METHOD copyCmds : BOOL
VAR_IN_OUT 
	r_slaveArmCtrlCmd :ST_SlaveArmCtrlCmds;
END_VAR
r_slaveArmCtrlCmd.m_jntEnableFlag :=m_jntEnableFlag;
r_slaveArmCtrlCmd.m_cmdCartPose:=m_cmdCartPose;
r_slaveArmCtrlCmd.m_cmdCartTwist:=m_cmdCartTwist;
r_slaveArmCtrlCmd.m_simJntPos:=m_simJntPos;
r_slaveArmCtrlCmd.m_cmdJntPos:=m_cmdJntPos;
r_slaveArmCtrlCmd.m_cmdJntVel:=m_cmdJntVel;
r_slaveArmCtrlCmd.m_cmdJntAcc:=m_cmdJntAcc;
r_slaveArmCtrlCmd.m_cmdJntTrq:=m_cmdJntTrq;
r_slaveArmCtrlCmd.m_jntOPMode:=m_jntOPMode;
r_slaveArmCtrlCmd.m_FFJntTrq:=m_FFJntTrq;
END_METHOD

// call this function to add friction compensation to m_cmdJntTrq
METHOD enableFrictionCompensation : BOOL
VAR_IN_OUT CONSTANT
	i_slaveArm :FB_SlaveArm;
END_VAR

VAR
	i:INT;
	frictionScale :LREAL;
END_VAR
// add joint friction compensation
FOR i:=1 TO g_sJntNum DO
	frictionScale :=LIMIT(-1.0, i_slaveArm.curJntVel[i]/g_fullFrictionVel,1.0);
	m_cmdJntTrq[i]:=m_cmdJntTrq[i]+frictionScale * g_frictionCompScale * GVL_SlaveArmDynamics.g_slaveJntFriction[i_slaveArm.armIdx, i];
END_FOR
END_METHOD

// override this function in each exact controller
// NOTICE: set joint control mode here, and do some initialization if needed
METHOD PUBLIC init : BOOL
VAR_IN_OUT CONSTANT
	i_slaveArm	:FB_SlaveArm;
END_VAR
VAR_IN_OUT 
	r_slaveArmCtrlCmd :ST_SlaveArmCtrlCmds;
END_VAR
m_timePeriod:=0;
m_jntEnableFlag :=g_onesVec8i;
m_jntOPMode:=g_slaveAllPosMode;
m_cmdCartPose:=i_slaveArm.curCartPose;
m_cmdCartTwist:=g_zeroVec6d;
IF FALSE = m_holdLastCmds THEN
	m_cmdJntPos:=i_slaveArm.curJntPos;
ELSE
	m_cmdJntPos:=r_slaveArmCtrlCmd.m_cmdJntPos;
END_IF
m_simJntPos := m_cmdJntPos;
m_cmdJntVel:=g_zeroVec8d;
m_cmdJntAcc:=g_zeroVec8d;
m_cmdJntTrq:=g_zeroVec8d;
m_FFJntTrq :=g_zeroVec8d;

// update commands to arm
copyCmds(r_slaveArmCtrlCmd);
END_METHOD

PROPERTY isFinished : BOOL
GET
isFinished:=m_isFinished;
END_GET
END_PROPERTY

{warning '添加方法实现'}
METHOD reset : BOOL
m_isFinished:=FALSE;
m_timePeriod:=0;
END_METHOD

{warning '添加方法实现'}
METHOD run : BOOL
VAR_IN_OUT CONSTANT
	i_endoscopePose : ST_Frame;
	i_masterStatus :ST_MasterStatus;
	i_setupStatus: ST_SetupStatus;
	i_slaveArm :FB_SlaveArm;
END_VAR
VAR_IN_OUT
	r_slaveArmCtrlCmd :ST_SlaveArmCtrlCmds;
END_VAR
VAR
	i:INT;
END_VAR
IF m_isFinished THEN
	RETURN;
END_IF

// check if arm enabled
IF FALSE = i_slaveArm.isEnabled(m_jntEnableFlag) THEN
	RETURN;
END_IF

// calculate command joint position--Motion control
calcCmdJntPos(i_endoscopePose, i_masterStatus, i_setupStatus, i_slaveArm);

// calculate command joint torque -- Force control
calcCmdJntTrq(i_endoscopePose, i_masterStatus, i_setupStatus, i_slaveArm);

// update commands to arm
copyCmds(r_slaveArmCtrlCmd);

// update time period
m_timePeriod := m_timePeriod+g_slaveArmCtrlCycleTime;
END_METHOD

PROPERTY timePeriod : Lreal
GET
timePeriod := m_timePeriod;
END_GET
END_PROPERTY

END_FUNCTION_BLOCK

// ---- FBs_SlaveControllers/FB_SlaveCtrlInit.TcPOU
// Brief: Slave Arm Init
FUNCTION_BLOCK PUBLIC FB_SlaveCtrlInit EXTENDS FB_SlaveArmCtrlBase
VAR_INPUT
END_VAR
VAR_OUTPUT
END_VAR
VAR
	m_initState :INT :=0;
	
	// SDO writer
	m_MotorCurrentSDOWrite: ARRAY[1..5] OF FB_EcCoESdoWrite;
	// power box joint motor rated current
	m_wristJntRatedCurrent : DINT := 200;
END_VAR

// override this function in each exact controller
METHOD PROTECTED calcCmdJntPos : BOOL
VAR_IN_OUT CONSTANT
	i_endoscopePose : ST_Frame;
	i_masterStatus :ST_MasterStatus;
	i_setupStatus: ST_SetupStatus;
	i_slaveArm :FB_SlaveArm;
END_VAR

VAR 
	jntIdx:INT;
	SDOSubIndexCur :WORD;
	armIdx:INT;
END_VAR
IF m_timePeriod > 1.0 THEN
	m_isFinished := TRUE;
END_IF

// reset instrument control box motor current limit
armIdx :=i_slaveArm.armIdx;
FOR jntIdx :=4 TO 8 DO
	//动力盒移动关节和器械旋转关节，共享一个控制字，由SDO写入
	IF (jntIdx=8)  THEN
		SDOSubIndexCur:=16#6098;
	//动力盒3、5号电机为一个驱动器，共享一个控制字，由SDO写入
	ELSIF (jntIdx=4) OR (jntIdx=6)  THEN
		SDOSubIndexCur:=16#6099;
	//动力盒2、4号电机为一个驱动器，共享一个控制字，由SDO写入
	ELSIF (jntIdx=5) OR (jntIdx=7)  THEN
		SDOSubIndexCur:=16#609A;
	END_IF

	// write max motor current if it changes and works in position mode  GVL_SlaveMotorParameters.g_motorMaxCurrent[jntIdx]
	m_MotorCurrentSDOWrite[jntIdx-3](sNetID:= GVL_SlaveJointEncoderCaliData.g_slaveArmNetID[armIdx],
					nSlaveAddr := GVL_SlaveJointEncoderCaliData.g_slaveJointNetPort[armIdx,jntIdx],
					nSubIndex:=0,nIndex:=SDOSubIndexCur,pSrcBuf:=ADR(m_wristJntRatedCurrent),
					cbBufLen:=SIZEOF(m_wristJntRatedCurrent),bExecute:=TRUE);
	IF NOT m_MotorCurrentSDOWrite[jntIdx-3].bBusy THEN
		m_MotorCurrentSDOWrite[jntIdx-3](bExecute:=FALSE);
	END_IF
	
END_FOR
END_METHOD

METHOD PUBLIC init : BOOL
VAR_IN_OUT CONSTANT
	i_slaveArm	:FB_SlaveArm;
END_VAR
VAR_IN_OUT 
	r_slaveArmCtrlCmd :ST_SlaveArmCtrlCmds;
END_VAR

VAR
	i:INT;
END_VAR
SUPER^.Init(i_slaveArm,r_slaveArmCtrlCmd);
m_jntEnableFlag:=g_zeroVec8i;

// update commands to arm
copyCmds(r_slaveArmCtrlCmd);
END_METHOD

END_FUNCTION_BLOCK

// ---- FBs_SlaveControllers/FB_SlaveCtrlSelfCheck.TcPOU
// Brief: Slave Arm Run Self-check Trajectory
FUNCTION_BLOCK PUBLIC FB_SlaveCtrlSelfCheck EXTENDS FB_SlaveArmCtrlBase
VAR CONSTANT
	m_selfCheckMotionNum :INT :=1;
END_VAR
VAR
	// slave self-check motion parameters
	m_selfCheckPosture:ARRAY [1..m_selfCheckMotionNum, 1..g_sJntNum] OF LREAL:=[0.0, 	-PI/2, GVL_SlaveMotorParameters.g_maxDHJntPos[3], 	5(-g_2pi)];																			//PI/4, -PI/4, 0.3, pi, pi, pi, pi, pi];
	m_selfCheckMaxjntVel:Vec8d:=[0.2, 0.2, 0.1, 5(2.0)];
	m_selfCheckMaxjntAcc:Vec8d:=[1.0, 1.0, 0.5, 5(4.0)];
	m_selfCheckMaxjntJerk:Vec8d:=[2.0,2.0, 1.0, 5(8.0)];
	
	m_selfCheckTrajIdx: INT := 1;
	m_slefCheckPlanner: ARRAY[1..m_selfCheckMotionNum] OF FB_TrajMoveJ;
	
   // wait time for joint enable
   m_enableWaitTime :LREAL := 1.0;

   // time gap between enable and motion
   m_jntMotionTimeGap :LREAL := 0.5;

	
END_VAR

// override this function in each exact controller
METHOD PROTECTED calcCmdJntPos : BOOL
VAR_IN_OUT CONSTANT
	i_endoscopePose : ST_Frame;
	i_masterStatus :ST_MasterStatus;
	i_setupStatus: ST_SetupStatus;
	i_slaveArm :FB_SlaveArm;
END_VAR

VAR 
	i :INT;
	curJntVel :Vec8d;
END_VAR
// check if planner is ready
IF m_slefCheckPlanner[m_selfCheckTrajIdx].isGene = FALSE THEN
	calcCmdJntPos:=FALSE;
	RETURN;
END_IF

// arms enable successively
IF m_timePeriod > m_enableWaitTime THEN
       m_jntEnableFlag :=g_onesVec8i;
END_IF

IF m_timePeriod < m_enableWaitTime + m_jntMotionTimeGap THEN
	RETURN;
END_IF

// traj plan
calcCmdJntPos :=m_slefCheckPlanner[m_selfCheckTrajIdx].evaluate(m_timePeriod-m_enableWaitTime-m_jntMotionTimeGap, jntPos=> m_cmdJntPos, jntVel=>m_cmdJntVel, jntAcc=> m_cmdJntAcc);

// check if to transit to next segment
curJntVel :=i_slaveArm.curJntVel;
IF(m_timePeriod - m_enableWaitTime - m_jntMotionTimeGap > m_slefCheckPlanner[m_selfCheckTrajIdx].duration  AND norm(curJntVel)<7*GVL_SlaveControlParameters.g_jntStaticVelThres) THEN
	m_selfCheckTrajIdx:=m_selfCheckTrajIdx+1;
	m_timePeriod:=0;
END_IF

// check if to terminated
IF(m_selfCheckTrajIdx > m_selfCheckMotionNum) THEN
	m_isFinished:=TRUE;
END_IF
END_METHOD

METHOD PUBLIC init : BOOL
VAR_IN_OUT CONSTANT
	i_slaveArm	:FB_SlaveArm;
END_VAR
VAR_IN_OUT 
	r_slaveArmCtrlCmd :ST_SlaveArmCtrlCmds;
END_VAR

VAR
	i,j :INT;
	startJntPos,endJntPos :Vec8d;
	baseJntPos:Vec8d;
	cycleNum :LREAL;
END_VAR
SUPER^.Init(i_slaveArm,r_slaveArmCtrlCmd);
//m_jntEnableFlag :=g_zeroVec8i;

//set different wait time for each arm, so the arms would run self-check successively
m_enableWaitTime := i_slaveArm.armIdx-1;

// determine base joint position for instrument joint
baseJntPos :=g_zeroVec8d;
FOR i:=4 TO g_sJntNum DO
	cycleNum := FLOOR(i_slaveArm.curJntPos[i]/g_2pi);
	baseJntPos[i]:=cycleNum* g_2Pi;
END_FOR

// traj plan
// fisrt segment
// TODO: joint1/2 stay still in case arms collision
m_selfCheckTrajIdx :=1;
startJntPos:=i_slaveArm.curJntPos;
endJntPos:=startJntPos;
FOR j:=3 TO g_sJntNum DO 
	endJntPos[j]:=baseJntPos[j]+m_selfCheckPosture[1,j];
END_FOR
m_slefCheckPlanner[1].init(startJntPos,endJntPos,m_selfCheckMaxjntVel, m_selfCheckMaxjntAcc,m_selfCheckMaxjntJerk);

// other segments
IF m_selfCheckMotionNum>= 2 THEN
	FOR i:=2 TO m_selfCheckMotionNum DO 
		FOR j:=1 TO 7 DO 
			startJntPos[j]:=baseJntPos[j]+m_selfCheckPosture[i-1,j];
			endJntPos[j]:=baseJntPos[j]+m_selfCheckPosture[i,j];
		END_FOR
		m_slefCheckPlanner[i].init(startJntPos,endJntPos,m_selfCheckMaxjntVel, m_selfCheckMaxjntAcc,m_selfCheckMaxjntJerk);
	END_FOR
END_IF;

// update commands to arm
copyCmds(r_slaveArmCtrlCmd);
END_METHOD

END_FUNCTION_BLOCK

// ---- FBs_TrajectoryPlanning/FB_TrajMoveJ.TcPOU
FUNCTION_BLOCK FB_TrajMoveJ EXTENDS FB_TrajBase
VAR_OUTPUT
END_VAR
VAR
	// move vector in joint space
	m_startPos:Vec8d;
	m_targetPos:Vec8d;
	m_moveDir : Vec8d;
	m_moveDistance :LREAL;
	
	// doubleS planning for move distance
	m_doubleS :FB_BasicDoubleS;
END_VAR

METHOD evaluate : BOOL
VAR_INPUT
	t :LREAL;
END_VAR

VAR_OUTPUT
	jntPos,jntVel, jntAcc :vec8d;
END_VAR
VAR
	q,q_dot,q_ddot :LREAL;
	moveRange :Vec8d;
END_VAR
evaluate:=m_doubleS.evaluate(t,q=>q,q_dot=>q_dot, q_ddot=>q_dot);
IF evaluate =FALSE THEN
	RETURN;
END_IF

vecMultiNum(m_moveDir,q, moveRange);
vecAdd(moveRange, m_startPos,jntPos);
vecMultiNum(m_moveDir,q_dot, jntVel);
vecMultiNum( m_moveDir,q_ddot, jntAcc);
END_METHOD

METHOD init : BOOL
VAR_INPUT
	i_startJntPos :Vec8d;
	i_targetJntPos :Vec8d;
	i_maxJntVel : Vec8d;
	i_maxJntAcc : Vec8d;
	i_maxJntJerk :Vec8d;
END_VAR
VAR 
	i:INT;
	maxV, maxA, maxJ :LREAL;
	q:ARRAY[1..2] OF LREAL;
	v:ARRAY[1..2] OF LREAL;
END_VAR
m_startPos:=i_startJntPos;
m_targetPos:=i_targetJntPos;
vecSub(i_targetJntPos, i_startJntPos, m_moveDir);
m_moveDistance := norm(m_moveDir);

IF(m_moveDistance<g_smallNum) THEN
	vecMultiNum(g_onesVec7d,1/8, m_moveDir);;
ELSE
	vecMultiNum( m_moveDir,1/m_moveDistance, m_moveDir);
END_IF

// determian max vel/acc/jerk
maxV:=g_largeNum;
maxA:=g_largeNum;
maxJ:=g_largeNum;
FOR i :=1 TO 7 DO 
	IF ABS(m_moveDir[i])>g_smallNum THEN
		maxV := MIN (maxV, ABS(i_maxJntVel[i]/m_moveDir[i]));
		maxA := MIN (maxA, ABS(i_maxJntAcc[i]/m_moveDir[i]));
		maxJ := MIN (maxJ, ABS(i_maxJntJerk[i]/m_moveDir[i]));
	END_IF
END_FOR

// planning for moving distance
q[1]:=0;
q[2]:=m_moveDistance;
v[1]:=0;
v[2]:=0;
m_doubleS.init(q,v, maxV, maxA, maxJ);
m_duration:=m_doubleS.duration;
m_isGenerated:=m_doubleS.isGene;
END_METHOD

END_FUNCTION_BLOCK

// ---- FBs_SlaveControllers/FB_SlaveCtrlStandBy.TcPOU
// Brief: Slave Arm Standby
FUNCTION_BLOCK PUBLIC FB_SlaveCtrlStandBy EXTENDS FB_SlaveArmCtrlBase
VAR_INPUT
END_VAR
VAR_OUTPUT
END_VAR
VAR
END_VAR

METHOD PUBLIC init : BOOL
VAR_IN_OUT CONSTANT
	i_slaveArm	:FB_SlaveArm;
END_VAR
VAR_IN_OUT 
	r_slaveArmCtrlCmd :ST_SlaveArmCtrlCmds;
END_VAR
//init
SUPER^.Init(i_slaveArm,r_slaveArmCtrlCmd);
END_METHOD

END_FUNCTION_BLOCK

// ---- FBs_SlaveControllers/FB_SlaveCtrlMountPanel.TcPOU
// Brief: Mounting Panel
FUNCTION_BLOCK PUBLIC FB_SlaveCtrlMountPanel EXTENDS FB_SlaveArmCtrlBase
VAR_INPUT
END_VAR
VAR_OUTPUT
END_VAR
VAR
	// mount status
	m_mountStatus :INT := 0;
	
	// flag if joint is mounted
	m_jointMounted :ARRAY[1..5] OF BOOL := [5(FALSE)];
	
	// mount motion planning
	m_jntOTG :ARRAY[1..5] OF FB_secOrdTrajFilter;
	m_panelMountVel :LREAL := 2*pi;
	m_panelMountAcc :LREAL := 4*pi;
	
	// joint current threshold which indicate motor is buckled with panel
	m_maxJntCurrent :INT := 80;
	
	// command mount motion
	m_mountStepPos :LREAL := 45.0 * g_deg2Rad;
	m_targetMountPos :Vec5d;
	
	//panel clamp error Id
	m_panelClampErrId : UINT;
	m_panelClampTime : LREAL;
	m_noCurrentTime : LREAL :=10;
	m_notReturnToZero : LREAL :=15;
END_VAR

// override this function in each exact controller
METHOD PROTECTED calcCmdJntPos : BOOL
VAR_IN_OUT CONSTANT
	i_endoscopePose : ST_Frame;
	i_masterStatus :ST_MasterStatus;
	i_setupStatus: ST_SetupStatus;
	i_slaveArm :FB_SlaveArm;
END_VAR

VAR 
	i :INT;
	curJntPos :Vec8d;
	jntPosErr :Vec8d;
	cycleNum :LREAL;
END_VAR
IF m_panelClampErrId>0 THEN
	RETURN;
END_IF

curJntPos := i_slaveArm.curJntPos;

CASE m_mountStatus OF
	// To lock joint with panel
	0:
		FOR i:=1 TO 5 DO
			// check joint buckled with panel
			IF ABS(i_slaveArm.filtJntCurrent[i+3])> m_maxJntCurrent THEN 
				m_jointMounted[i]:=TRUE;
				m_targetMountPos[i]:=curJntPos[i+3];
				m_jntOTG[i].init(m_targetMountPos[i], 0,m_panelMountVel, m_panelMountAcc, g_slaveArmCtrlCycleTime);
			END_IF
			
			// set command joint position step
			IF FALSE = m_jointMounted[i] THEN
				m_targetMountPos[i]:=curJntPos[i+3]+m_mountStepPos;
			END_IF
		END_FOR
		
		IF (m_jointMounted[1] AND m_jointMounted[2] AND m_jointMounted[3] AND m_jointMounted[4] AND m_jointMounted[5]) or m_timePeriod > 5.0 THEN
			m_mountStatus:=1;
		END_IF
	
	// determine zero position
	1:
		FOR i:=1 TO 5 DO
			cycleNum := FLOOR(curJntPos[i+3]/g_2pi);
			m_targetMountPos[i]:=cycleNum* g_2Pi;
		END_FOR
		m_mountStatus :=2;
	
	// move back to zero position
	2:
		m_isFinished:=TRUE;
		FOR i:=1 TO 5 DO
			IF ABS(m_targetMountPos[i]-curJntPos[i+3])>GVL_SlaveControlParameters.g_jntCtrlAngTolHigh THEN
				m_isFinished:=FALSE;
				EXIT;
			END_IF
		END_FOR
END_CASE

//panel clamp status check
m_panelClampErrId := panelClampStatus();

// traj plan
FOR i:=1 TO 5 DO
	m_jntOTG[i].run(m_targetMountPos[i],0.0, o_cmdAcc=>m_cmdJntAcc[3+i],o_cmdVel=>m_cmdJntVel[3+i],o_cmdPos=>m_cmdJntPos[i+3]);
END_FOR
END_METHOD

METHOD PUBLIC init : BOOL
VAR_IN_OUT CONSTANT
	i_slaveArm	:FB_SlaveArm;
END_VAR
VAR_IN_OUT 
	r_slaveArmCtrlCmd :ST_SlaveArmCtrlCmds;
END_VAR
VAR
	i : INT;
END_VAR
SUPER^.Init(i_slaveArm,r_slaveArmCtrlCmd);
m_jntOPMode[4] := DriverOPMode_PosTrq;
m_jntOPMode[5] := DriverOPMode_PosTrq;
m_jntOPMode[6] := DriverOPMode_PosTrq;
m_jntOPMode[7] := DriverOPMode_PosTrq;
m_jntOPMode[8] := DriverOPMode_PosTrq;

m_mountStatus:=0;
FOR i:=1 TO 5 DO
	m_targetMountPos[i]:=m_cmdJntPos[i+3];
	m_jntOTG[i].init(m_targetMountPos[i], 0,m_panelMountVel, m_panelMountAcc, g_slaveArmCtrlCycleTime);
	m_jointMounted[i]:=FALSE;
END_FOR
m_panelClampTime :=0;
m_panelClampErrId := 0;
// update commands to arm
copyCmds(r_slaveArmCtrlCmd);
END_METHOD

PROPERTY panelClampErrId : UINT
GET
panelClampErrId := m_panelClampErrId;
END_GET
END_PROPERTY

METHOD panelClampStatus : UINT
VAR_IN_OUT CONSTANT
END_VAR
//m_panelClampErrId=1 panel clamp the current does not reach the set value
//m_panelClampErrId=2 panel clamp position does not return to zero
m_panelClampTime := LIMIT(0,m_panelClampTime + g_slaveArmCtrlCycleTime,10);

IF m_mountStatus=0  AND m_panelClampTime>=m_noCurrentTime  THEN
	panelClampStatus := 1;
ELSIF m_mountStatus=2 AND m_panelClampTime>=m_notReturnToZero  THEN
	panelClampStatus := 2;
END_IF
END_METHOD

END_FUNCTION_BLOCK

// ---- FBs_SlaveControllers/FB_SlaveCtrlPanelReady.TcPOU
// Brief: Panel Ready
FUNCTION_BLOCK PUBLIC FB_SlaveCtrlPanelReady EXTENDS FB_SlaveArmCtrlBase
VAR_INPUT
END_VAR
VAR_OUTPUT
END_VAR
VAR
END_VAR

// override this function in each exact controller
// NOTICE: set joint control mode here, and do some initialization if needed
METHOD PUBLIC init : BOOL
VAR_IN_OUT CONSTANT
	i_slaveArm	:FB_SlaveArm;
END_VAR
VAR_IN_OUT 
	r_slaveArmCtrlCmd :ST_SlaveArmCtrlCmds;
END_VAR
//init
SUPER^.Init(i_slaveArm,r_slaveArmCtrlCmd);

//update the control mode ---1028
m_jntOPMode := g_slaveAllPosMode;
m_jntOPMode[1]:=DriverOPMode_PosTrq;
m_jntOPMode[2]:=DriverOPMode_PosTrq;

copyCmds(r_slaveArmCtrlCmd);
END_METHOD

END_FUNCTION_BLOCK

// ---- FBs_SlaveControllers/FB_SlaveCtrlMountInstru.TcPOU
// Brief: Mounting Instrument
FUNCTION_BLOCK PUBLIC FB_SlaveCtrlMountInstru EXTENDS FB_SlaveArmCtrlBase
VAR
	// mount status
	m_instruMountStatus :INT := 0;
	m_scopeMountStatus :INT := 0;
	m_ultrasoundMountStatus :INT :=0 ;
	
	// flag if joint is mounted
	m_jointMounted :ARRAY[1..5] OF BOOL := [5(FALSE)];
	
	// instrument mount motion range
	m_mountMotionAng :Vec5d :=[5(pi)];
	
	// instrument mount direction
	m_mountDir :Vec5i :=[1, 1, 1, 1, 1];
	
	// mount motion planning
	m_jntOTG :ARRAY[1..5] OF FB_secOrdTrajFilter;
	m_instruMountVel :LREAL := 4*PI;
	m_instruMountAcc :LREAL := 8*PI;
	
	//Joint 4 half-range angle of instrument
	m_instruJnt4HalfRangeAng :LREAL := 323*g_deg2Rad;
	
	// joint current threshold which indicate panel is buckled with instrument
	m_maxJntCurrent :Vec5d := [150, 150, 150, 180, 180];
	
	// command mount motion
	m_targetMountPos :Vec8d;
	
	// instrument zero position
	m_instruZeroDeviation :Vec5d;
	
	//ultrasound knife Reduce the current rotation Angle  J3
	m_ultraKnifeRotaAngleJ3 :LREAL := 30*g_deg2Rad;
	
	// ultrasound knife rotate angle zero position
	m_ultraKnifeRotAngZeroPos :LREAL := 4.50567;
	
	// joint position error
	m_jntPosErr :Vec5d;
	
	// endoscope motion angle to original position
	m_scopeJnt4CenterMotionAng :LREAL :=175*g_deg2Rad;
	m_scopeJnt5CenterMotionAng :LREAL :=150*g_deg2Rad;
	
	//instrument clamp error Id
	m_instruClampErrId : UINT;
	m_instruClampTime : LREAL;
	m_noCurrentTime : LREAL :=3;
	m_notReturnToZero : LREAL :=5;
END_VAR

// override this function in each exact controller
METHOD PROTECTED calcCmdJntPos : BOOL
VAR_IN_OUT CONSTANT
	i_endoscopePose : ST_Frame;
	i_masterStatus :ST_MasterStatus;
	i_setupStatus: ST_SetupStatus;
	i_slaveArm :FB_SlaveArm;
END_VAR

VAR 
END_VAR
// mount error detect;
m_instruClampErrId := instruClampStatus(i_slaveArm);

// return directly if instrument/endoscope is not readed
IF NOT(i_slaveArm.instrument.onChipData.m_InstruReadSucceed) THEN
	return;
END_IF

IF i_slaveArm.instrument.onChipData.m_InstruReadSucceed AND InstruType_endoscope = i_slaveArm.instrument.onChipData.m_InstruID THEN
	mountEndoscope(i_slaveArm);
ELSIF i_slaveArm.instrument.onChipData.m_InstruReadSucceed AND InstruType_NewEndoscope = i_slaveArm.instrument.onChipData.m_InstruID THEN
	mountNewEndoscope(i_slaveArm);
ELSIF i_slaveArm.instrument.onChipData.m_InstruReadSucceed AND (InstruType_UltrasoundKnifeS = i_slaveArm.instrument.m_instruType OR InstruType_UltrasoundKnifeU = i_slaveArm.instrument.m_instruType) THEN
	mountUltraKnife(i_slaveArm);
ELSE
	mountInstrument(i_slaveArm);
END_IF
END_METHOD

METHOD PUBLIC init : BOOL
VAR_IN_OUT CONSTANT
	i_slaveArm	:FB_SlaveArm;
END_VAR
VAR_IN_OUT 
	r_slaveArmCtrlCmd :ST_SlaveArmCtrlCmds;
END_VAR

VAR
	i : INT;
END_VAR
// check if to hold the command joint position unchanged
m_holdLastCmds := checkToHoldLastCmds(i_slaveArm);

SUPER^.Init(i_slaveArm,r_slaveArmCtrlCmd);
m_jntOPMode[4] := DriverOPMode_PosTrq;
m_jntOPMode[5] := DriverOPMode_PosTrq;
m_jntOPMode[6] := DriverOPMode_PosTrq;
m_jntOPMode[7] := DriverOPMode_PosTrq;
m_jntOPMode[8] := DriverOPMode_PosTrq;

FOR i:=1 TO 5 DO
	m_targetMountPos[i+3]:=m_cmdJntPos[i+3];
	m_jntOTG[i].init(m_targetMountPos[i+3], 0,m_instruMountVel, m_instruMountAcc, g_slaveArmCtrlCycleTime);
	m_jointMounted[i]:=FALSE;
END_FOR

m_instruMountStatus:=0;
m_scopeMountStatus:=0;
m_ultrasoundMountStatus:=0;
m_instruClampErrId := 0;
m_instruClampTime := 0;
// update commands to arm
copyCmds(r_slaveArmCtrlCmd);
END_METHOD

PROPERTY instruClampErrId :  UINT
GET
instruClampErrId := m_instruClampErrId;
END_GET
END_PROPERTY

METHOD instruClampStatus : UINT
VAR_IN_OUT CONSTANT
	i_slaveArm :FB_SlaveArm;
END_VAR
//m_instruClampErrId=1 instrumen clamp the current does not reach the set value
//m_instruClampErrId=2 instrumen clamp position does not return to zero
m_instruClampTime := LIMIT(0,m_instruClampTime + g_slaveArmCtrlCycleTime,10);
IF i_slaveArm.instrument.onChipData.m_InstruReadSucceed THEN
	IF InstruType_endoscope = i_slaveArm.instrument.m_instruType THEN
		IF (m_scopeMountStatus=0 OR m_scopeMountStatus=1) AND m_instruClampTime>=m_noCurrentTime  THEN
			instruClampStatus := 1;
		ELSIF m_scopeMountStatus=3 AND m_instruClampTime>=m_notReturnToZero  THEN
			instruClampStatus := 2;
		END_IF
		
	ELSIF (InstruType_UltrasoundKnifeS = i_slaveArm.instrument.m_instruType OR InstruType_UltrasoundKnifeU = i_slaveArm.instrument.m_instruType) THEN
		IF (m_ultrasoundMountStatus=0) AND m_instruClampTime>=m_noCurrentTime  THEN
			instruClampStatus := 1;
		ELSIF (m_scopeMountStatus=3) AND m_instruClampTime>=m_notReturnToZero  THEN
			instruClampStatus := 2;
		END_IF
			
	ELSE
		IF (m_instruMountStatus=0) AND m_instruClampTime>=m_noCurrentTime  THEN
			instruClampStatus := 1;
		ELSIF (m_instruMountStatus=3) AND m_instruClampTime>=m_notReturnToZero  THEN
			instruClampStatus := 2;
		END_IF
	END_IF
END_IF
END_METHOD

METHOD mountEndoscope : BOOL
VAR_IN_OUT CONSTANT
	i_slaveArm :FB_SlaveArm;
END_VAR

VAR 
	i :INT;
	curJntPos :Vec8d;
END_VAR
curJntPos := i_slaveArm.curJntPos;

CASE m_scopeMountStatus OF
	//fix scope lock joint(joint 7)
	0:
		// other joints stay still
		FOR i:=1 TO 3 DO
			m_jointMounted[i] := TRUE;
			m_targetMountPos[i+3]:=curJntPos[i+3];
			m_jntOTG[i].init(m_targetMountPos[i+3], 0,m_instruMountVel, m_instruMountAcc, g_slaveArmCtrlCycleTime);
		END_FOR
	
		// check if buckled
		m_jointMounted[4]:=FALSE; 
		m_jointMounted[5]:=FALSE; 
		IF ABS(i_slaveArm.filtJntCurrent[7])> m_maxJntCurrent[4] THEN 
			m_jointMounted[4]:=TRUE;
			m_targetMountPos[7]:=curJntPos[7];
			m_jntOTG[4].init(m_targetMountPos[7], 0,m_instruMountVel, m_instruMountAcc, g_slaveArmCtrlCycleTime);
			m_scopeMountStatus:=1;
		ELSE
			m_targetMountPos[7]:=curJntPos[7]+m_mountMotionAng[4];
		END_IF

	1: // buckle scope rotate joint (joint 8)
		m_jointMounted[5]:=FALSE; 
		IF ABS(i_slaveArm.filtJntCurrent[8])> m_maxJntCurrent[5] THEN 
			m_jointMounted[5]:=TRUE;
			m_targetMountPos[8]:=curJntPos[8];
			m_jntOTG[5].init(m_targetMountPos[8], 0,m_instruMountVel, m_instruMountAcc, g_slaveArmCtrlCycleTime);
			m_scopeMountStatus:=2;
		ELSE
			m_targetMountPos[8]:=curJntPos[8]+m_mountMotionAng[5];
		END_IF
	

	2:// move back to zero position
		m_targetMountPos[7]:= curJntPos[7]-m_scopeJnt4CenterMotionAng;
		m_targetMountPos[8]:= curJntPos[8]-m_scopeJnt5CenterMotionAng;
		m_scopeMountStatus :=3;
		
		
	3:
		IF ABS(m_targetMountPos[7]-curJntPos[7]) <GVL_SlaveControlParameters.g_jntCtrlAngTolHigh AND 
				ABS(m_targetMountPos[8]-curJntPos[8]) <GVL_SlaveControlParameters.g_jntCtrlAngTolHigh THEN
			// record current joint position as offset for instrument
			i_slaveArm.instrument.initInstruJntPos(i_slaveArm.curJntPos);
			m_isFinished := TRUE;
		END_IF
		
END_CASE

// traj plan
FOR i:=1 TO 5 DO
	m_jntOTG[i].run(m_targetMountPos[i+3],0.0, o_cmdAcc=>m_cmdJntAcc[3+i],o_cmdVel=>m_cmdJntVel[3+i],o_cmdPos=>m_cmdJntPos[i+3]);
END_FOR
END_METHOD

METHOD mountInstrument : BOOL
VAR_IN_OUT CONSTANT
	i_slaveArm :FB_SlaveArm;
END_VAR

VAR 
	i :INT;
	curJntPos :Vec8d;
END_VAR
curJntPos := i_slaveArm.curJntPos;

// joint4 stay still if instrument has only on finger
IF i_slaveArm.instrument.instruTypeInfo.m_isSingleFinger THEN
	m_jointMounted[1]:=TRUE;
END_IF

CASE m_instruMountStatus OF
	// To lock panel with instrument
	0:
		//buckle panel with instrument
		FOR i:=1 TO 4 DO
			// check if buckled 
			IF ABS(i_slaveArm.filtJntCurrent[i+3])> m_maxJntCurrent[i] AND ABS(i_slaveArm.curJntVel[i+3])<1.0*g_deg2Rad THEN 
				m_jointMounted[i]:=TRUE;
				m_targetMountPos[i+3]:=curJntPos[i+3];
				m_jntOTG[i].init(m_targetMountPos[i+3], 0,m_instruMountVel, m_instruMountAcc, g_slaveArmCtrlCycleTime);
			END_IF
			
			// set target joint position
			IF FALSE = m_jointMounted[i] THEN
				IF i = 4 THEN
					m_targetMountPos[i+3]:=curJntPos[i+3]+m_mountMotionAng[i];
				ELSE
					m_targetMountPos[i+3]:=curJntPos[i+3]-m_mountMotionAng[i];
				END_IF
				
			END_IF
		END_FOR
		
		
		// check transition condition
		IF (m_jointMounted[1] AND m_jointMounted[2] AND m_jointMounted[3] AND m_jointMounted[4])  THEN
			IF i_slaveArm.instrument.onChipData.m_InstruReadSucceed THEN//Check whether the data is read successfully
				m_instruMountStatus:=1;
			END_IF
		END_IF
	
	1:// calculation deviates from the instrument zero position
		FOR i:=1 TO 4 DO
			m_instruZeroDeviation[i] :=  i_slaveArm.linkSingle[i+3] - i_slaveArm.instrument.onChipData.m_InstruPos[i];
		END_FOR
		m_instruMountStatus :=2;
	
	
	2:// move back to zero position
		FOR i:=1 TO 3 DO//J1-3
			IF m_instruZeroDeviation[i]>pi THEN
				m_instruZeroDeviation[i] := m_instruZeroDeviation[i] - 2*PI;
			ELSIF m_instruZeroDeviation[i]<-pi THEN
				m_instruZeroDeviation[i] := m_instruZeroDeviation[i] + 2*PI;
			END_IF
		END_FOR
		
		//joint4
		IF m_instruZeroDeviation[4]>0 AND m_instruZeroDeviation[4] < pi THEN
			m_instruZeroDeviation[4] := m_instruZeroDeviation[4] - 2*pi;
		ELSIF m_instruZeroDeviation[4]<0 AND m_instruZeroDeviation[4] > -pi THEN
			m_instruZeroDeviation[4] := m_instruZeroDeviation[4] + 2*pi;
		END_IF
		
		// set target joint position
		FOR i:=1 TO 4 DO
			m_targetMountPos[i+3]:=curJntPos[i+3] - m_instruZeroDeviation[i];
		END_FOR
		m_instruMountStatus :=3;
	
	3: // move to zero position
		m_instruMountStatus :=4;
		FOR i:=1 TO 4 DO 
			m_jntPosErr[i]:=m_targetMountPos[i+3]-curJntPos[i+3];
			IF ABS(m_jntPosErr[i]) >GVL_SlaveControlParameters.g_jntCtrlAngTolLow OR 
					ABS( i_slaveArm.linkSingle[i+3] - i_slaveArm.instrument.onChipData.m_InstruPos[i]) >5*g_deg2rad THEN
				m_instruMountStatus :=3;
				EXIT;
			END_IF
		END_FOR
	
	4:
		// record current joint position as offset for instrument
		i_slaveArm.instrument.initInstruJntPos(i_slaveArm.curJntPos);
		
		m_isFinished :=  TRUE;

END_CASE

// traj plan
FOR i:=1 TO 4 DO
	m_jntOTG[i].run(m_targetMountPos[i+3],0.0, o_cmdAcc=>m_cmdJntAcc[3+i],o_cmdVel=>m_cmdJntVel[3+i],o_cmdPos=>m_cmdJntPos[i+3]);
END_FOR
END_METHOD

METHOD mountNewEndoscope : BOOL
VAR_IN_OUT CONSTANT
	i_slaveArm :FB_SlaveArm;
END_VAR

VAR 
	i :INT;
	curJntPos :Vec8d;
END_VAR
curJntPos := i_slaveArm.curJntPos;

CASE m_scopeMountStatus OF
	//fix scope lock joint(joint 7)
	0:
		// other joints stay still
		FOR i:=1 TO 5 DO
			IF i = 1 OR i =2 OR i =5 THEN
				m_jointMounted[i] := TRUE;
				m_targetMountPos[i+3]:=curJntPos[i+3];
				m_jntOTG[i].init(m_targetMountPos[i+3], 0,m_instruMountVel, m_instruMountAcc, g_slaveArmCtrlCycleTime);
			END_IF
		END_FOR
	
		// check if buckled
		m_jointMounted[3]:=FALSE; 
		m_jointMounted[4]:=FALSE; 
		FOR i:=3 TO 4 DO
			IF ABS(i_slaveArm.filtJntCurrent[i+3])> m_maxJntCurrent[i] THEN 
				m_jointMounted[i]:=TRUE;
				m_targetMountPos[i+3]:=curJntPos[i+3];
				m_jntOTG[i].init(m_targetMountPos[i+3], 0,m_instruMountVel, m_instruMountAcc, g_slaveArmCtrlCycleTime);
				
			ELSE
				m_targetMountPos[i+3]:=curJntPos[i+3]+m_mountMotionAng[i];
			END_IF
		END_FOR
		
		IF m_jointMounted[3] AND m_jointMounted[4] THEN
			m_scopeMountStatus:=1;
		END_IF
		

	1: // buckle scope rotate joint (joint 8)
		m_jntOPMode[6] := DriverOPMode_Trq;
		m_instruZeroDeviation[4] :=  i_slaveArm.linkSingle[7] - i_slaveArm.instrument.onChipData.m_InstruPos[4];
		m_scopeMountStatus :=2;

	2:// move back to zero position
		
		//joint4
		IF m_instruZeroDeviation[4]>0 AND m_instruZeroDeviation[4] > pi THEN
			m_instruZeroDeviation[4] := m_instruZeroDeviation[4] - 2*pi;
		ELSIF m_instruZeroDeviation[4]<0 AND m_instruZeroDeviation[4] < -pi THEN
			m_instruZeroDeviation[4] := m_instruZeroDeviation[4] + 2*pi;
		END_IF
		
		m_targetMountPos[7]:=curJntPos[7] - m_instruZeroDeviation[4];
		m_scopeMountStatus :=3;
		
		
	3:
		m_isFinished := FALSE;
		IF ABS(m_targetMountPos[7]-curJntPos[7]) <GVL_SlaveControlParameters.g_jntCtrlAngTolHigh THEN
			// record current joint position as offset for instrument
			i_slaveArm.instrument.initInstruJntPos(i_slaveArm.curJntPos);
			m_isFinished := TRUE;
		END_IF
		
END_CASE

// traj plan
FOR i:=1 TO 5 DO
	m_jntOTG[i].run(m_targetMountPos[i+3],0.0, o_cmdAcc=>m_cmdJntAcc[3+i],o_cmdVel=>m_cmdJntVel[3+i],o_cmdPos=>m_cmdJntPos[i+3]);
END_FOR

// joint6 output torque to help rotation motion
IF m_jntOPMode[6] = DriverOPMode_Trq THEN
	m_cmdJntTrq[6] := -0.5*i_slaveArm.cmdJntTrq[7];
END_IF
END_METHOD

METHOD mountUltraKnife : BOOL
VAR_IN_OUT CONSTANT
	i_slaveArm :FB_SlaveArm;
END_VAR

VAR 
	i :INT;
	curJntPos :Vec8d;
END_VAR
curJntPos := i_slaveArm.curJntPos;

m_jointMounted[1]:=TRUE;
m_jointMounted[2]:=TRUE;


CASE m_ultrasoundMountStatus OF 
	// To lock panel with instrument
	0:
		//buckle panel with instrument
		FOR i:=3 TO 5 DO
			// check if buckled 
			IF ABS(i_slaveArm.filtJntCurrent[i+3])> m_maxJntCurrent[i] THEN 
				m_jointMounted[i]:=TRUE;
				m_targetMountPos[i+3]:=curJntPos[i+3];
				m_jntOTG[i].init(m_targetMountPos[i+3], 0,m_instruMountVel, m_instruMountAcc, g_slaveArmCtrlCycleTime);
			END_IF
			
			// set target joint position
			IF FALSE = m_jointMounted[i] THEN
				IF i = 5 THEN
					m_targetMountPos[i+3]:=curJntPos[i+3]+m_mountMotionAng[i];
				ELSE
					m_targetMountPos[i+3]:=curJntPos[i+3]-m_mountMotionAng[i];
				END_IF
				
			END_IF
		END_FOR

		// check transition condition
		IF ( m_jointMounted[3] AND m_jointMounted[4] AND m_jointMounted[5] )  THEN
			IF i_slaveArm.instrument.onChipData.m_InstruReadSucceed THEN//Check whether the data is read successfully
				m_ultrasoundMountStatus:=1;
			END_IF
		END_IF

	1:
		//m_jntOPMode[8] := DriverOPMode_Trq;
		// calculation deviates from the instrument zero position
		m_instruZeroDeviation[3] :=   i_slaveArm.linkSingle[6] - i_slaveArm.instrument.onChipData.m_InstruPos[3]; //m_ultraKnifeRotaAngleJ3;
		m_instruZeroDeviation[4] :=  i_slaveArm.linkSingle[7] - m_ultraKnifeRotAngZeroPos;
		m_ultrasoundMountStatus :=2;
		
	2:// move back to zero position
		//joint3
		IF m_instruZeroDeviation[3] > 2*pi THEN
			m_instruZeroDeviation[3] := m_instruZeroDeviation[3] - 2*pi  ;
		ELSIF  m_instruZeroDeviation[3] < -pi THEN
			m_instruZeroDeviation[3] := 2*pi + m_instruZeroDeviation[3] ;
		END_IF
		//joint4
		IF m_instruZeroDeviation[4]>0 AND m_instruZeroDeviation[4] < pi THEN
			m_instruZeroDeviation[4] := m_instruZeroDeviation[4] - 2*pi;
		ELSIF m_instruZeroDeviation[4]<0 AND m_instruZeroDeviation[4] > -pi THEN
			m_instruZeroDeviation[4] := m_instruZeroDeviation[4] + 2*pi;
		END_IF
	
		// set target joint position
		m_targetMountPos[6]:=curJntPos[6] - m_instruZeroDeviation[3];
		m_targetMountPos[7]:=curJntPos[7] - m_instruZeroDeviation[4];
		m_targetMountPos[8]:=curJntPos[8] - m_instruZeroDeviation[4];

		m_ultrasoundMountStatus :=3;

	3:
		// joint8 in passive mode
		m_jntOPMode[8] := DriverOPMode_Trq;
		
		m_isFinished:=TRUE;
		FOR i:=3 TO 4 DO 
			m_jntPosErr[i]:=m_targetMountPos[i+3]-curJntPos[i+3];
			IF ABS(m_jntPosErr[i]) >GVL_SlaveControlParameters.g_jntCtrlAngTolLow  THEN
				m_isFinished := FALSE;
				EXIT;
			END_IF
		END_FOR	
		
		// record current joint position as offset for instrument
		i_slaveArm.instrument.initInstruJntPos(i_slaveArm.curJntPos);

END_CASE


// traj plan
FOR i:=1 TO 5 DO
	m_jntOTG[i].run(m_targetMountPos[i+3],0.0, o_cmdAcc=>m_cmdJntAcc[3+i],o_cmdVel=>m_cmdJntVel[3+i],o_cmdPos=>m_cmdJntPos[i+3]);
END_FOR
END_METHOD

END_FUNCTION_BLOCK

// ---- FBs_SlaveControllers/FB_SlaveCtrlInstruReady.TcPOU
// Brief: Instrument Ready
FUNCTION_BLOCK PUBLIC FB_SlaveCtrlInstruReady EXTENDS FB_SlaveArmCtrlBase
VAR_INPUT
END_VAR
VAR_OUTPUT
END_VAR
VAR
END_VAR

METHOD PUBLIC init : BOOL
VAR_IN_OUT CONSTANT
	i_slaveArm	:FB_SlaveArm;
END_VAR
VAR_IN_OUT 
	r_slaveArmCtrlCmd :ST_SlaveArmCtrlCmds;
END_VAR


VAR
	j:INT;
	maxJntErr:LREAL;
	jntCtrlErr:Vec7d;
END_VAR
//NOTE:DO NOT hold last command

//init
SUPER^.Init(i_slaveArm,r_slaveArmCtrlCmd);
END_METHOD

END_FUNCTION_BLOCK

// ---- FBs_SlaveControllers/FB_SlaveCtrlMasterSlave.TcPOU
// Brief: Slave Arm MasterSlave controller
FUNCTION_BLOCK PUBLIC FB_SlaveCtrlMasterSlave EXTENDS FB_SlaveArmCtrlBase
VAR
	// pose track control kp
	m_posTrackKp :REAL := 0;
	m_oriTrackKp :REAL := 100;
	
	// minimum distance between instrument tip and remote center
	m_minInstruRCDis:LREAL := 0.05;
	
	// master-slave motion scale
	m_MSMotionScale :LREAL;
		
	// gripper match angle threshold
	m_gripperMatchAngThres :LREAL := 2*g_deg2Rad;
	
	// control error thershold from joint limit back to free space
	m_jntLimitOriErr :LREAL :=g_deg2Rad * 5;
	
	// master-slave error thershold to halt control 
	m_safetyOriErr :LREAL :=g_deg2Rad * 150;
	
	// filter cut-off frequency for master-slave control
	m_macroCmdJntPosLpfCutoffFreq : LREAL :=5;
	m_microCmdJntPosLpfCutoffFreq : LREAL :=15;
	
	// last command joint position
	m_lastCmdJntPos :Vec8d;
	
	// simulated DH joint position
	m_simDHJntPos : Vec6d;
	
	// simulated slave twist of DH joint
	m_simDHJointVel :Vec6d;
		
	// enter master-slave control for the first time
	m_firstIn :BOOL := TRUE;
	
	// flag if reach joint limit
	m_reachMacroJntLimit :BOOL;
	m_reachWristJntLimit :BOOL;
	m_jntLimitFlag :Vec6b;
	
	// master/slave origin pose when first enter master-slave control
	m_masterOriginPose : ST_Frame;
	m_slaveOriginPose : ST_Frame;
	
	// orientation deviation(in master coordinate) between master and slave when first enter control
	m_MSOriDeviation : Mat3d;
	
	// command joint position filter
	m_cmdJntPosLpf:ARRAY[1..8] OF FB_LowPassFilter;
	
	// commmand yaw angle and velocity
	m_cmdYawAngle :LREAL;
	m_cmdYawVel :LREAL;
	
	// comand yaw angle and velocity filter
	m_cmdYawAngLpf : FB_LowPassFilter;
	m_cmdYawVelLpf : FB_LowPassFilter;
	
	// master pose/velocity in monitor coordinate
	m_masterPose :ST_Frame;
	m_masterTwist : Vec6d;
	
	// master grip angle
	m_masterGripAngle : LREAL;
	
	// slave command/current pose in endoscope coordinate
	m_slaveCmdPoseInScope :ST_Frame;
	m_slavePoseInScope : ST_Frame;
	
	// slave command/current pose in cart
	m_slaveCmdPoseInCart :ST_Frame;
	m_slavePoseInCart : ST_Frame;
	
	// instrument controller
	m_basicInstruController : FB_BasicInstruControl;
	m_usKnifeController : FB_UltrosonicKnifeControl;
	
	// slave command grip angle and grip force level
	m_slaveCmdGripAngle :LREAL;
	m_slaveCmdGripForceLevel:LREAL;
	
	// slave pose error
	m_slavePosErr :Vec3d;
	m_slaveRotErr :Mat3d;
	m_errAngle : LREAL;
	m_errAxisLocal, m_errAxis :Vec3d;
	m_masterSlavePoseError :Vec6d;
	
	// master velocity in slave coordinate
	m_masterFFVel, m_masterFFWVel :Vec3d;
	
	// velocity for slave to track master motion
	m_slaveCmdVel, m_slaveCmdWVel : Vec3d;
	
	// flag to start gripper control
	m_gripperCtrlFlag :BOOL;
	
	// instrument tyep
	m_instruType : E_InstrumentType;
	
	//################# variable to interpolate master pose ##############
	m_firstInterpolate :BOOL :=TRUE;
	m_lastMasterPose : ST_Frame;
	m_lastMasterGripAngle :LREAL;
	m_masterInterpolateCycle :INT := 4;
	m_curInterpolateCylce :INT := 1;
	m_masterPosInterStep :Vec3d;
	m_masterOriInterStep :Mat3d;
	m_masterGripAngleInterStep :LREAL;
	m_interplotedMasterPose :ST_Frame;
	m_interplotedMasterGripAngle :LREAL;
	
	// code execute time measure
	m_codeTime : Profiler;
	
	
END_VAR

METHOD PROTECTED calcCmdJntPos : BOOL
VAR_IN_OUT CONSTANT
	i_endoscopePose : ST_Frame;
	i_masterStatus :ST_MasterStatus;
	i_setupStatus: ST_SetupStatus;
	i_slaveArm :FB_SlaveArm;
END_VAR

VAR 
	i,j : INT;
	tmpMat3d : Mat3d;
	masterMotionRange : Vec3d;
	
	masterVelInScope, masterWVelInScope :Vec3d;
	masterVelInCart, masterWVelInCart :Vec3d;

	cmdVelScale :LREAL;
	invJaco :Mat6d;
	armJntJaco,armJntJacoInv, wristJntJaco :Mat3d;
	velByWristJnt,velByArmJnt : Vec3d;
	armDHJntVel, wristDHJntVel :Vec3d;
	tmpFrame : ST_Frame;
	jnt3Limit :LREAL;
	jntDynaUB, jntDynaLB :LREAL;
END_VAR
m_codeTime(START:=TRUE, RESET:=TRUE);

IF isFinished THEN
	RETURN;
END_IF

// decide matched master arm index
FOR i:=1 TO g_mArmNum DO 
	IF i_masterStatus.m_teleSlaveArmIdx[i] = i_slaveArm.armIdx THEN
		masterPoseInterploate(i_masterStatus.m_curArmPose[i],i_masterStatus.m_gripAngle[i], i_slaveArm);
		m_masterPose := m_interplotedMasterPose;
		m_masterGripAngle := m_interplotedMasterGripAngle;
		m_masterTwist := i_masterStatus.m_curArmTwist[i];
	END_IF
END_FOR

// compute slave pose in endoscope coordinate
m_slavePoseInCart := transform(i_setupStatus.m_curEndPose[i_slaveArm.armIdx], i_slaveArm.simCartPose);
tmpFrame :=invFrame(i_endoscopePose);
m_slavePoseInScope := transform(tmpFrame, m_slavePoseInCart);

// handle for the first time in
IF TRUE = m_firstIn THEN
	m_firstIn := FALSE;
	m_masterOriginPose :=m_masterPose;
	m_slaveOriginPose := m_slavePoseInScope;
	matTranspose(m_masterOriginPose.m_rot, tmpMat3d);
	matMultiply(tmpMat3d, m_slavePoseInScope.m_rot,m_MSOriDeviation);
	m_lastMasterGripAngle := m_masterGripAngle;
	
	// only update motion scale while entering teleControl 
	m_MSMotionScale := 1.0/ MAX(1,  i_masterStatus.m_motionScale);
END_IF

// compute master twist in slave arm coordinate
FOR i:=1 TO 3 DO
	masterVelInScope[i] := m_masterTwist[i]*m_MSMotionScale;
	masterWVelInScope[i] := m_masterTwist[i+3];
END_FOR
matMultiVec(i_endoScopePose.m_rot, masterVelInScope, masterVelInCart);
matMultiVec(i_endoScopePose.m_rot, masterWVelInScope, masterWVelInCart);
matTranspose(i_setupStatus.m_curEndPose[i_slaveArm.armIdx].m_rot, tmpMat3d);
matMultiVec(tmpMat3d,masterVelInCart, m_masterFFVel);
matMultiVec(tmpMat3d,masterWVelInCart, m_masterFFWVel);

// compute slave command pose in scope
vecSub(m_masterPose.m_pos, m_masterOriginPose.m_pos, masterMotionRange);
vecSelfMultiNum(masterMotionRange, m_MSMotionScale);
vecAdd(m_slaveOriginPose.m_pos, masterMotionRange, m_slaveCmdPoseInScope.m_pos);
matMultiply(m_masterPose.m_rot, m_MSOriDeviation, m_slaveCmdPoseInScope.m_rot);

// compute slave command pose in slave arm coordinate
m_slaveCmdPoseInCart := transform(i_endoScopePose, m_slaveCmdPoseInScope);
tmpFrame := invFrame(i_setupStatus.m_curEndPose[i_slaveArm.armIdx]);
m_cmdCartPose := transform(tmpFrame, m_slaveCmdPoseInCart);

// compute pose error
vecSub(m_cmdCartPose.m_pos, i_slaveArm.simCartPose.m_pos, m_slavePosErr);
matTranspose(i_slaveArm.simCartPose.m_rot, tmpMat3d);
matMultiply(tmpMat3d, m_cmdCartPose.m_rot, m_slaveRotErr);
rot2AngAxis(m_slaveRotErr, angle=>m_errAngle, axis=>m_errAxisLocal);
matMultiVec(i_slaveArm.simCartPose.m_rot, m_errAxisLocal, m_errAxis);

// calculate pose error in endoscope
calcMSErrInScope(i_endoscopePose, i_setupStatus.m_curEndPose[i_slaveArm.armIdx], i_slaveArm);

//safety check
IF ABS(m_errAngle)>m_safetyOriErr THEN
	m_isFinished := TRUE;
	RETURN;
END_IF

// pose track control
vecMultiNum(m_slavePosErr, m_posTrackKp, m_slaveCmdVel);
vecMultiNum(m_errAxis, m_errAngle*m_oriTrackKp, m_slaveCmdWVel);
// final command twist
FOR i:=1 TO 3 DO 
	m_cmdCartTwist[i] := m_slaveCmdVel[i] + m_masterFFVel[i];
	m_cmdCartTwist[i+3] := m_slaveCmdWVel[i] + m_masterFFWVel[i];
END_FOR

// compute command velocity for DH joints
invJaco := i_slaveArm.simJacoInv;
matMultiVec(invJaco, m_cmdCartTwist, m_simDHJointVel);

// limit instrument wrist dofs
limitInstruDofs(i_slaveArm, m_simDHJointVel);

// limit instrument wrist joint velocity
wristLimitSolve(i_slaveArm);

// limit DH joints velocity 
FOR i:=4 TO 6 DO 
	m_simDHJointVel[i] := LIMIT(-GVL_SlaveMotorParameters.g_maxJntVel[i], m_simDHJointVel[i], GVL_SlaveMotorParameters.g_maxJntVel[i]);
END_FOR

// modify arm joints velocity to compensate wrist joint motion
FOR i:=1 TO 3 DO
	FOR j:=1 TO 3 DO
		armJntJaco[i,j]:=i_slaveArm.simJaco[i,j];
		wristJntJaco[i,j]:=i_slaveArm.simJaco[i,j+3];
	END_FOR
	armDHJntVel[i]:=m_simDHJointVel[i];
	wristDHJntVel[i]:=m_simDHJointVel[i+3];
	m_slaveCmdVel[i] := m_cmdCartTwist[i];
END_FOR
invMat3(armJntJaco, armJntJacoInv);
matMultiVec(wristJntJaco, wristDHJntVel, velByWristJnt);
vecSub(m_slaveCmdVel, velByWristJnt, velByArmJnt);
matMultiVec(armJntJacoInv, velByArmJnt, armDHJntVel);

// limit arm joint position
m_reachMacroJntLimit:=false;
FOR i:=1 TO 3 DO
	IF i=3 THEN
		jnt3Limit := i_slaveArm.instrument.instruTypeInfo.m_rodLength+i_slaveArm.instrument.instruTypeInfo.m_headLength - GVL_SlaveArmKinematic.g_minInstruRCDis;
		jntDynaUB := MAX( 0, (jnt3Limit - i_slaveArm.simDHJntPos[i])/g_slaveArmCtrlCycleTime);
	ELSE
		jntDynaUB := MAX( 0, (GVL_SlaveMotorParameters.g_maxDHJntPos[i] - i_slaveArm.simDHJntPos[i])/g_slaveArmCtrlCycleTime);
	END_IF
	jntDynaLB := MIN( 0, (GVL_SlaveMotorParameters.g_minDHJntPos[i] - i_slaveArm.simDHJntPos[i])/g_slaveArmCtrlCycleTime);
	
	IF m_simDHJointVel[i] >= jntDynaUB OR m_simDHJointVel[i]<= jntDynaLB THEN
		armDHJntVel[i]:=LIMIT(jntDynaLB, m_simDHJointVel[i], jntDynaUB);
		m_reachMacroJntLimit:=TRUE;
	END_IF
END_FOR

// limit DH joints velocity 
FOR i:=1 TO 3 DO
	m_simDHJointVel[i]:=armDHJntVel[i];
	m_simDHJointVel[i+3]:=wristDHJntVel[i];
END_FOR
cmdVelScale := 1;
FOR i:=1 TO g_cartDofs DO 
	cmdVelScale:=MAX(cmdVelScale, ABS(m_simDHJointVel[i]/GVL_SlaveMotorParameters.g_maxJntVel[i]));
END_FOR
vecSelfMultiNum(m_simDHJointVel, 1.0/cmdVelScale);

// integrate command DH joint position
FOR i:=1 TO 6 DO
	m_simDHJntPos[i] := i_slaveArm.simDHJntPos[i] + m_simDHJointVel[i]*g_slaveArmCtrlCycleTime;
END_FOR

// gripper angle/force control
gripperControl(i_slaveArm);

// calculate target motor joint position/velocity from DH joint position
i_slaveArm.instrument.instruIK(m_simDHJntPos,m_slaveCmdGripAngle, o_jntPos=>m_simJntPos);

// filt command joint position
FOR i:=1 TO g_sJntNum DO 
	m_cmdJntPos[i] := m_cmdJntPosLpf[i].run(m_simJntPos[i]);
END_FOR

// compute command joint velocity
vecSub(m_cmdJntPos, m_lastCmdJntPos, m_cmdJntVel);
vecSelfMultiNum(m_cmdJntVel, g_slaveArmCtrlFreq);
m_lastCmdJntPos:=m_cmdJntPos;

m_codeTime(START:=FALSE);
END_METHOD

// override this function in each exact controller
METHOD PROTECTED calcCmdJntTrq : BOOL
VAR_IN_OUT CONSTANT
	i_endoscopePose : ST_Frame;
	i_masterStatus :ST_MasterStatus;
	i_setupStatus: ST_SetupStatus;
	i_slaveArm :FB_SlaveArm;
END_VAR
VAR
	i :INT ;
	instruCmdGripAngle, instruCmdGripForceLevel :LREAL;
	instruCmdJntPos, instruCmdJntVel : Vec5d;	
	instruJntCtrlTrq :Vec5d;
END_VAR
IF isFinished THEN
	RETURN;
END_IF

// set joint torque to zero in default
m_cmdJntTrq := g_zeroVec8d;

// instrument joint control
FOR i:=1 TO 5 DO 
	instruCmdJntPos[i]:=m_cmdJntPos[i+3];
	instruCmdJntVel[i]:=m_cmdJntVel[i+3];
END_FOR
m_cmdYawAngle := m_cmdYawAngLpf.run(m_simDHJntPos[6]);
m_cmdYawVel := m_cmdYawVelLpf.run(m_simDHJointVel[6]);

// check if to exert larger grip force
setMaxGripTrq(i_masterStatus, i_slaveArm);


IF i_slaveArm.instrument.instruType = InstruType_UltrasoundKnifeS OR i_slaveArm.instrument.instruType = InstruType_UltrasoundKnifeU THEN
	m_usKnifeController.run(instruCmdJntPos,instruCmdJntVel, m_slaveCmdGripForceLevel, i_slaveArm, o_cmdJntTrq=>instruJntCtrlTrq);
ELSE
	m_basicInstruController.run(instruCmdJntPos,instruCmdJntVel, m_cmdYawAngle, m_cmdYawVel, m_slaveCmdGripForceLevel, i_slaveArm, o_cmdJntTrq=>instruJntCtrlTrq);
END_IF

FOR i:=1 TO 5 DO
	m_cmdJntTrq[i+3]:=instruJntCtrlTrq[i];
END_FOR
END_METHOD

METHOD calcMSErrInScope : BOOL
VAR_IN_OUT CONSTANT
	i_endoscopePose : ST_Frame;
	i_setupPose :ST_Frame;
	i_slaveArm :FB_SlaveArm;
END_VAR
VAR
	posErrInCart,oriErrInCart :Vec3d;
	invRot :Mat3d;
	posErrInScope,oriErrInScope :Vec3d;
	i:INT;
END_VAR
m_masterSlavePoseError := g_zeroVec6d;

// pose error caused by joints limits
IF m_reachMacroJntLimit THEN
	// pose error in cart coordinate
	matMultiVec(i_setupPose.m_rot, m_slavePosErr, posErrInCart);
	
	// pose err in endoscope coordinate
	matTranspose(i_endoscopePose.m_rot, invRot);
	matMultiVec(invRot, posErrInCart, posErrInScope);
	
	FOR i:=1 TO 3 DO 
		m_masterSlavePoseError[i]:=posErrInScope[i];
	END_FOR
END_IF

// pose error caused by joints limits
IF  m_reachWristJntLimit THEN
	// pose error in cart coordinate
	matMultiVec(i_setupPose.m_rot, m_errAxis, oriErrInCart);
	vecSelfMultiNum(oriErrInCart, m_errAngle);
	
	// pose err in endoscope coordinate
	matTranspose(i_endoscopePose.m_rot, invRot);
	matMultiVec(invRot, oriErrInCart, oriErrInScope);
	
	FOR i:=1 TO 3 DO 
		m_masterSlavePoseError[i+3]:=oriErrInScope[i];
	END_FOR
END_IF
END_METHOD

METHOD PUBLIC clearBacklash : BOOL
VAR_INPUT
END_VAR
m_basicInstruController.clearBacklash();
m_usKnifeController.clearBacklash();
END_METHOD

METHOD gripperControl : BOOL
VAR_IN_OUT CONSTANT
	i_slaveArm :FB_SlaveArm;
END_VAR

VAR
	matchedSlaveGripAngle:LREAL;
	matchedSlaveGripForce:LREAL;
	masterGripVelThres :LREAL := 5.0 *g_deg2Rad;
END_VAR
// compute matched slave grip angle and force
i_slaveArm.instrument.gripAngleMap(m_masterGripAngle,o_instruGripAngle=>matchedSlaveGripAngle, o_instruGripForceLevel=>matchedSlaveGripForce);

IF m_gripperCtrlFlag THEN
	m_slaveCmdGripAngle := matchedSlaveGripAngle;
	m_slaveCmdGripForceLevel := matchedSlaveGripForce;
	RETURN;
ELSE
	//m_gripperCtrlFlag := (ABS(m_masterGripAngleVel) >masterGripVelThres) AND  (m_masterGripAngleVel * (matchedSlaveGripAngle-i_slaveArm.curGripAngle)>0);
	m_gripperCtrlFlag := ABS(matchedSlaveGripAngle-i_slaveArm.curGripAngle)<m_gripperMatchAngThres OR 
	     (matchedSlaveGripAngle>=i_SlaveArm.instrument.instruTypeInfo.m_maxGripAngle - m_gripperMatchAngThres AND i_slaveArm.curGripAngle>=matchedSlaveGripAngle) OR 
		(matchedSlaveGripAngle<=g_minSlaveGripAngle + m_gripperMatchAngThres AND i_slaveArm.curGripAngle<=matchedSlaveGripAngle);
END_IF
END_METHOD

METHOD PUBLIC init : BOOL
VAR_IN_OUT CONSTANT
	i_slaveArm	:FB_SlaveArm;
END_VAR
VAR_IN_OUT 
	r_slaveArmCtrlCmd :ST_SlaveArmCtrlCmds;
END_VAR
VAR 
	i :INT ;
END_VAR
SUPER^.Init(i_slaveArm,r_slaveArmCtrlCmd);
m_simJntPos :=m_cmdJntPos;
m_lastCmdJntPos :=m_cmdJntPos;
m_jntOPMode[1] := DriverOPMode_PosTrq;
m_jntOPMode[2] := DriverOPMode_PosTrq;
m_jntOPMode[3] := DriverOPMode_PosTrq;
m_jntOPMode[4] := DriverOPMode_Trq;
m_jntOPMode[5] := DriverOPMode_Trq;
m_jntOPMode[6] := DriverOPMode_Trq;
m_jntOPMode[7] := DriverOPMode_Trq;
m_jntOPMode[8] := DriverOPMode_Trq;
m_firstIn :=TRUE;
m_gripperCtrlFlag :=FALSE;

// init gripper angle
m_slaveCmdGripAngle := i_slaveArm.curGripAngle;
m_slaveCmdGripForceLevel:=0;

// init filter
FOR i:=1 TO 3 DO
	m_cmdJntPosLpf[i].init(1, m_macroCmdJntPosLpfCutoffFreq, g_slaveArmCtrlFreq);
END_FOR
FOR i:=4 TO g_sJntNum DO
	m_cmdJntPosLpf[i].init(1, m_microCmdJntPosLpfCutoffFreq, g_slaveArmCtrlFreq);
END_FOR
m_cmdYawAngLpf.init(1, m_microCmdJntPosLpfCutoffFreq, g_slaveArmCtrlFreq);
m_cmdYawVelLpf.init(1, m_microCmdJntPosLpfCutoffFreq, g_slaveArmCtrlFreq);

// init controller
m_basicInstruController.init(i_slaveArm);
m_usKnifeController.init(i_slaveArm);
m_instruType := i_slaveArm.instrument.instruType;

// init interpolation data
m_firstInterpolate :=TRUE;
m_curInterpolateCylce := 1;

// update commands to arm
copyCmds(r_slaveArmCtrlCmd);
END_METHOD

PROPERTY InstruBacklash : Vec5d
GET
IF m_instruType = InstruType_UltrasoundKnifeS OR m_instruType = InstruType_UltrasoundKnifeU THEN
	instruBacklash := m_usKnifeController.m_jntBacklash;
ELSE
	instruBacklash := m_basicInstruController.m_jntBacklash;
END_IF
END_GET
END_PROPERTY

// limit specific joint dofs based on instrument types
METHOD PRIVATE limitInstruDofs : BOOL
VAR_IN_OUT CONSTANT
	i_slaveArm :FB_SlaveArm;
END_VAR

VAR_IN_OUT
	r_simDHJointVel :Vec6d;
END_VAR
IF i_slaveArm.instrument.instruType = InstruType_UltrasoundKnifeS OR i_slaveArm.instrument.instruType = InstruType_UltrasoundKnifeU THEN
	r_simDHJointVel[5] :=0;
	r_simDHJointVel[6] :=0;
END_IF
END_METHOD

// every some cycles the data from master robots would be miss, so add this interpolation
METHOD masterPoseInterploate : BOOL
VAR_IN_OUT CONSTANT
	i_masterPose :ST_FRAME;
	i_masterGripAngle :LREAL;
	i_slaveArm :FB_SlaveArm;
END_VAR

VAR
	rotT :Mat3d;
	rotErr:Mat3d;
	errAngle:LREAL;
	errAxisLocal :Vec3d;
	tmpMat :Mat3d;
	cartVel, DHJntVel :Vec6d;
	wVelWrd:Vec3d;
	i :INT;
	invJaco :Mat6d;
	cmdVelScale :LREAL;
END_VAR
IF m_firstInterpolate THEN
	m_firstInterpolate :=FALSE;
	m_lastMasterGripAngle :=i_masterGripAngle;
	m_lastMasterPose := i_masterPose;
	m_masterPosInterStep :=g_zeroVec3d;
	m_masterOriInterStep :=g_eye3d;
	m_masterGripAngleInterStep :=0.0;
	m_interplotedMasterPose := i_masterPose;
	m_interplotedMasterGripAngle := i_masterGripAngle;
END_IF


// update next interpolation
IF m_curInterpolateCylce > m_masterInterpolateCycle THEN
	vecSub(i_masterPose.m_pos, m_lastMasterPose.m_pos, m_masterPosInterStep);
	vecSelfMultiNum( m_masterPosInterStep, 1.0/INT_TO_LREAL(m_masterInterpolateCycle));
	
	matTranspose(m_lastMasterPose.m_rot, rotT);
	matMultiply(rotT, i_masterPose.m_rot, rotErr);
	rot2AngAxis(rotErr, angle=>errAngle, axis=>errAxisLocal);
	m_masterOriInterStep := angAxis2Rot(errAngle/INT_TO_LREAL(m_masterInterpolateCycle), errAxisLocal);
	
	// cap linear step based on macro joint velocity limit
	matMultiVec(i_slaveArm.simCartPose.m_rot, errAxisLocal, wVelWrd);
	vecSelfMultiNum(wVelWrd, errAngle*g_slaveArmCtrlFreq/INT_TO_LREAL(m_masterInterpolateCycle));
	FOR i:=1 TO 3 DO
		cartVel[i] := m_masterPosInterStep[i]*m_MSMotionScale*g_slaveArmCtrlFreq;
		cartVel[i+3] := wVelWrd[i];
	END_FOR
	invJaco := i_slaveArm.simJacoInv;
	matMultiVec(invJaco, cartVel, DHJntVel);
	cmdVelScale := 1;
	FOR i:=1 TO 3 DO 
		cmdVelScale:=MAX(cmdVelScale, ABS(DHJntVel[i]/GVL_SlaveMotorParameters.g_maxJntVel[i]));
	END_FOR
	vecSelfMultiNum(m_masterPosInterStep, 1.0/cmdVelScale);
	
	m_masterGripAngleInterStep := (i_masterGripAngle- m_lastMasterGripAngle)/INT_TO_LREAL(m_masterInterpolateCycle);
	
	m_curInterpolateCylce :=1;
	m_lastMasterPose:= i_masterPose;
	m_lastMasterGripAngle := i_masterGripAngle;
END_IF

// control points
IF m_curInterpolateCylce = m_masterInterpolateCycle THEN
	m_interplotedMasterGripAngle := m_lastMasterGripAngle;
	m_interplotedMasterPose.m_rot := m_lastMasterPose.m_rot;
ELSE
	m_interplotedMasterGripAngle := m_interplotedMasterGripAngle + m_masterGripAngleInterStep;
	vecSelfAdd(m_interplotedMasterPose.m_pos, m_masterPosInterStep);
	tmpMat := m_interplotedMasterPose.m_rot;
	matMultiply(tmpMat, m_masterOriInterStep, m_interplotedMasterPose.m_rot);
END_IF

m_curInterpolateCylce:= m_curInterpolateCylce+1;
END_METHOD

PROPERTY masterSlavePoseErr : REFERENCE to Vec6d
GET
masterSlavePoseErr REF= m_masterSlavePoseError;
END_GET
END_PROPERTY

METHOD setMaxGripTrq : BOOL
VAR_IN_OUT CONSTANT
	i_masterStatus :ST_MasterStatus;
	i_slaveArm :FB_SlaveArm;
END_VAR
VAR
	i:INT;
	 peakGripTrqScale :LREAL := 2;
END_VAR
// only valid for ForceBipolar
IF i_slaveArm.instrument.instruType <> InstruType_ForceBipolar THEN
	RETURN;
END_IF

// only trigger grip force switch when no grip force exerted currently
IF m_slaveCmdGripForceLevel > g_smallNum  THEN
	RETURN;
END_IF; 

// decide matched master arm index
FOR i:=1 TO g_mArmNum DO 
	IF i_masterStatus.m_teleSlaveArmIdx[i] = i_slaveArm.armIdx THEN
		IF i_masterStatus.m_pedalHover[i] AND i_masterStatus.m_electricKnifePedalTrigger[i] =1 THEN
		   m_basicInstruController.setMaxGripTrq(i_slaveArm.instrument.instruTypeInfo.m_normGripTrq * peakGripTrqScale);
		ELSE
		   m_basicInstruController.setMaxGripTrq(i_slaveArm.instrument.instruTypeInfo.m_normGripTrq);
		END_IF
	END_IF
END_FOR
END_METHOD

// calculate optimized wrist joint velocity when joint limit is violated
METHOD wristLimitSolve : BOOL
VAR_IN_OUT CONSTANT
	i_slaveArm :FB_SlaveArm;
END_VAR

VAR
	i,j:INT;
	jntDynaUB, jntDynaLB :LREAL;
	
	dsrWVel:Vec3d;
	wristJntVel :Vec3d;
	wristJaco:Mat3d;
	
	optJntVel:Vec2d;
	partJaco :Mat32;
	partJacoT :Mat23;
	JtJ,JtJInv :Mat2d;
	partJacoPInv:Mat23;
	
	partJacoPinv2 :Vec3d;
	jacoNorm :LREAL;
	
	wVelLocal,wVelWrd:Vec3d;
	matT:Mat3d;
END_VAR
m_reachWristJntLimit := FALSE;

// desire angular velocity from wrist joint
FOR i:=1 TO 3 DO
	wristJntVel[i] := m_simDHJointVel[i+3];
	FOR j:=1 TO 3 DO
		wristJaco[i,j]:= i_slaveArm.simJaco[i+3, j+3];
	END_FOR 
END_FOR
matMultiVec(wristJaco, wristJntVel, dsrWVel);

// check which joint reaches limit
FOR i:=4 TO 6 DO
	m_jntLimitFlag[i] := FALSE;
	jntDynaUB := MAX( 0, (i_slaveArm.instrument.m_wristMaxDHJntPos[i-3] - i_slaveArm.simDHJntPos[i])/g_slaveArmCtrlCycleTime);
	jntDynaLB := MIN( 0, (i_slaveArm.instrument.m_wristMinDHJntPos[i-3] - i_slaveArm.simDHJntPos[i])/g_slaveArmCtrlCycleTime);
	IF m_simDHJointVel[i] >= jntDynaUB OR m_simDHJointVel[i]<=jntDynaLB THEN
		m_simDHJointVel[i]:=LIMIT(jntDynaLB, m_simDHJointVel[i], jntDynaUB);
		m_jntLimitFlag[i]:=TRUE;
		m_reachWristJntLimit := TRUE;
	END_IF
END_FOR

// no limit violated
IF NOT( m_jntLimitFlag[4]) AND NOT(m_jntLimitFlag[5]) AND NOT(m_jntLimitFlag[6]) THEN
	RETURN;
END_IF; 

// all joint reach limit
IF m_jntLimitFlag[4] AND m_jntLimitFlag[5] AND m_jntLimitFlag[6] THEN
	RETURN;
END_IF;

// joint 4 reach limit
IF m_jntLimitFlag[4] AND NOT(m_jntLimitFlag[5]) AND NOT(m_jntLimitFlag[6]) THEN
	// colume 2/3
	partJaco[1,1]:= wristJaco[1,2];
	partJaco[2,1]:= wristJaco[2,2];
	partJaco[3,1]:= wristJaco[3,2];
	
	partJaco[1,2]:= wristJaco[1,3];
	partJaco[2,2]:= wristJaco[2,3];
	partJaco[3,2]:= wristJaco[3,3];
	
	// pinv partJaco
	matTranspose(partJaco, partJacoT);
	matMultiply(partJacoT, partJaco, JtJ);
	IF NOT(invMat2(JtJ, JtJInv)) THEN
		m_simDHJointVel[5] :=0;
		m_simDHJointVel[6] := 0;
		RETURN;
	END_IF
	matMultiply(JtJInv, partJacoT, partJacoPinv);
	
	// desire angular velocity exclusive limited joint motion
	dsrWVel[1] := dsrWVel[1] - wristJaco[1,1] * m_simDHJointVel[4];
	dsrWVel[2] := dsrWVel[2] - wristJaco[2,1] * m_simDHJointVel[4];
	dsrWVel[3] := dsrWVel[3] - wristJaco[3,1] * m_simDHJointVel[4];
	
	//NOTE: special handle for roll limit. avoiding joint5/6 motion caused by roll limit
	matTranspose(i_slaveArm.simCartPose.m_rot, matT);
	matMultiVec(matT, dsrWVel, wVelLocal);
	wVelLocal[3]:=0;
	matMultiVec(i_slaveArm.simCartPose.m_rot, wVelLocal, dsrWVel);
	
	// solve
	matMultiVec(partJacoPinv, dsrWVel, optJntVel);
	m_simDHJointVel[5] :=optJntVel[1];
	m_simDHJointVel[6] := optJntVel[2];
END_IF

// joint 5 reach limit
IF m_jntLimitFlag[5] AND NOT(m_jntLimitFlag[4]) AND NOT(m_jntLimitFlag[6]) THEN
	// colume 1/3
	partJaco[1,1]:= wristJaco[1,1];
	partJaco[2,1]:= wristJaco[2,1];
	partJaco[3,1]:= wristJaco[3,1];
	
	partJaco[1,2]:= wristJaco[1,3];
	partJaco[2,2]:= wristJaco[2,3];
	partJaco[3,2]:= wristJaco[3,3];
	
	// pinv partJaco
	matTranspose(partJaco, partJacoT);
	matMultiply(partJacoT, partJaco, JtJ);
	IF NOT(invMat2(JtJ, JtJInv)) THEN
		m_simDHJointVel[4] :=0;
		m_simDHJointVel[6] := 0;
		RETURN;
	END_IF
	matMultiply(JtJInv, partJacoT, partJacoPinv);
		
	// desire angular velocity exclusive limited joint motion
	dsrWVel[1] := dsrWVel[1] - wristJaco[1,2] * m_simDHJointVel[5];
	dsrWVel[2] := dsrWVel[2] - wristJaco[2,2] * m_simDHJointVel[5];
	dsrWVel[3] := dsrWVel[3] - wristJaco[3,2] * m_simDHJointVel[5];
	
	//NOTE: special handle for pitch limit. avoiding joint4/6 motion caused by pitch limit
	matTranspose(i_slaveArm.simCartPose.m_rot, matT);
	matMultiVec(matT, dsrWVel, wVelLocal);
	wVelLocal[1]:=0;
	matMultiVec(i_slaveArm.simCartPose.m_rot, wVelLocal, dsrWVel);
	
	// solve
	matMultiVec(partJacoPinv, dsrWVel, optJntVel);
	m_simDHJointVel[4] :=optJntVel[1];
	m_simDHJointVel[6] := optJntVel[2];
END_IF

// joint 6 reach limit
IF m_jntLimitFlag[6] AND NOT(m_jntLimitFlag[4]) AND NOT(m_jntLimitFlag[5]) THEN
	// colume 1/2
	partJaco[1,1]:= wristJaco[1,1];
	partJaco[2,1]:= wristJaco[2,1];
	partJaco[3,1]:= wristJaco[3,1];
	
	partJaco[1,2]:= wristJaco[1,2];
	partJaco[2,2]:= wristJaco[2,2];
	partJaco[3,2]:= wristJaco[3,2];
	
	// pinv partJaco
	matTranspose(partJaco, partJacoT);
	matMultiply(partJacoT, partJaco, JtJ);
	IF NOT(invMat2(JtJ, JtJInv)) THEN
		m_simDHJointVel[4] :=0;
		m_simDHJointVel[5] := 0;
		RETURN;
	END_IF
	matMultiply(JtJInv, partJacoT, partJacoPinv);
		
	// desire angular velocity exclusive limited joint motion
	dsrWVel[1] := dsrWVel[1] - wristJaco[1,3] * m_simDHJointVel[6];
	dsrWVel[2] := dsrWVel[2] - wristJaco[2,3] * m_simDHJointVel[6];
	dsrWVel[3] := dsrWVel[3] - wristJaco[3,3] * m_simDHJointVel[6];
	
	// solve
	matMultiVec(partJacoPinv, dsrWVel, optJntVel);
	m_simDHJointVel[4] :=optJntVel[1];
	m_simDHJointVel[5] := optJntVel[2];
END_IF

// joint 4/5 reach limit
IF m_jntLimitFlag[4] AND m_jntLimitFlag[5] AND NOT(m_jntLimitFlag[6]) THEN
	// pinv partJaco of column 3
	partJacoPinv2[1] := wristJaco[1, 3];
	partJacoPinv2[2] := wristJaco[2, 3];
	partJacoPinv2[3] := wristJaco[3, 3];
	jacoNorm := norm(partJacoPinv2);
	vecSelfMultiNum(partJacoPinv2, 1.0/(jacoNorm*jacoNorm));
		
	// desire angular velocity exclusive limited joint motion
	dsrWVel[1] := dsrWVel[1] - wristJaco[1,1] * m_simDHJointVel[4] - wristJaco[1,2] * m_simDHJointVel[5];
	dsrWVel[2] := dsrWVel[2] - wristJaco[2,1] * m_simDHJointVel[4] - wristJaco[2,2] * m_simDHJointVel[5];
	dsrWVel[3] := dsrWVel[3] - wristJaco[3,1] * m_simDHJointVel[4] - wristJaco[3,2] * m_simDHJointVel[5];
	
	// solve
	m_simDHJointVel[6] := vecDot(partJacoPinv2, dsrWVel);
END_IF

// joint 4/6 reach limit
IF m_jntLimitFlag[4] AND m_jntLimitFlag[6] AND NOT(m_jntLimitFlag[5]) THEN
	// pinv partJaco of column 2
	partJacoPinv2[1] := wristJaco[1, 2];
	partJacoPinv2[2] := wristJaco[2, 2];
	partJacoPinv2[3] := wristJaco[3, 2];
	jacoNorm := norm(partJacoPinv2);
	vecSelfMultiNum(partJacoPinv2, 1.0/(jacoNorm*jacoNorm));
		
	// desire angular velocity exclusive limited joint motion
	dsrWVel[1] := dsrWVel[1] - wristJaco[1,1] * m_simDHJointVel[4] - wristJaco[1,3] * m_simDHJointVel[6];
	dsrWVel[2] := dsrWVel[2] - wristJaco[2,1] * m_simDHJointVel[4] - wristJaco[2,3] * m_simDHJointVel[6];
	dsrWVel[3] := dsrWVel[3] - wristJaco[3,1] * m_simDHJointVel[4] - wristJaco[3,3] * m_simDHJointVel[6];
	
	// solve
	m_simDHJointVel[5] := vecDot(partJacoPinv2, dsrWVel);
END_IF

// joint 5/6 reach limit
IF m_jntLimitFlag[5] AND m_jntLimitFlag[6] AND NOT(m_jntLimitFlag[4]) THEN
	// pinv partJaco of column 4
	partJacoPinv2[1] := wristJaco[1, 1];
	partJacoPinv2[2] := wristJaco[2, 1];
	partJacoPinv2[3] := wristJaco[3, 1];
	jacoNorm := norm(partJacoPinv2);
	vecSelfMultiNum(partJacoPinv2, 1.0/(jacoNorm*jacoNorm));
		
	// desire angular velocity exclusive limited joint motion
	dsrWVel[1] := dsrWVel[1] - wristJaco[1,2] * m_simDHJointVel[5] - wristJaco[1,3] * m_simDHJointVel[6];
	dsrWVel[2] := dsrWVel[2] - wristJaco[2,2] * m_simDHJointVel[5] - wristJaco[2,3] * m_simDHJointVel[6];
	dsrWVel[3] := dsrWVel[3] - wristJaco[3,2] * m_simDHJointVel[5] - wristJaco[3,3] * m_simDHJointVel[6];
	
	// solve
	m_simDHJointVel[4] := vecDot(partJacoPinv2, dsrWVel);
END_IF


// check which joint reaches limit
FOR i:=4 TO 6 DO
	jntDynaUB := MAX( 0, (i_slaveArm.instrument.m_wristMaxDHJntPos[i-3] - i_slaveArm.simDHJntPos[i])/g_slaveArmCtrlCycleTime);
	jntDynaLB := MIN( 0, (i_slaveArm.instrument.m_wristMinDHJntPos[i-3] - i_slaveArm.simDHJntPos[i])/g_slaveArmCtrlCycleTime);
	IF m_simDHJointVel[i] >= jntDynaUB OR m_simDHJointVel[i]<=jntDynaLB THEN
		m_simDHJointVel[i]:=LIMIT(jntDynaLB, m_simDHJointVel[i], jntDynaUB);
		m_jntLimitFlag[i]:=TRUE;
		m_reachWristJntLimit := TRUE;
	END_IF
END_FOR
END_METHOD

END_FUNCTION_BLOCK

// ---- FBs_BasicControllers/FB_BasicInstruControl.TcPOU
// instrument joints control
FUNCTION_BLOCK FB_BasicInstruControl
VAR_INPUT
END_VAR
VAR_OUTPUT
END_VAR
VAR
	// instrument PID control paramters
	m_instruKp:ARRAY[1..5] OF LREAL:=[4(5),0.0];
	m_instruKd:ARRAY[1..5] OF LREAL:=[4(0.25), 0];
	m_instruKi:ARRAY[1..5] OF LREAL:=[4(10.0),0];
	m_instruKiLimit:ARRAY[1..5] OF LREAL:=[5(50.0)];
	m_instruCtrlLimit:ARRAY[1..5] OF LREAL:=[2(120.0), 3(200.0)];
	
	// gripper force level threshold for variable PID parameter
	m_forceLevelThres : ARRAY[1..3] OF LREAL := [40, 70, 101];
	
	// yaw PID control (when fingers grasp with force)
	m_yawKp:ARRAY[1..3] OF LREAL:=[5, 8, 10];
	m_yawKd:ARRAY[1..3] OF LREAL:=[0.25, 0.4, 0.6];
	m_yawKi:ARRAY[1..3] OF LREAL:=[10.0, 15.0, 20.0];
	m_yawKiLimit:LREAL:=100.0;
	m_yawCtrlLimit:LREAL:=200.0;
	
	// max grip force/current(mA)
	m_maxGripForce:LREAL;
	m_maxGripCurrent:LREAL:=150.0;
	
	// max gripper finger control force/current(mA)
	m_maxGripCtrlForce:LREAL;
	m_maxGripCtrlCurrent:LREAL:=250.0;
	
	// ratio convert motor current to joint troque
	m_currentRatioMotor2Jnt:LREAL;
	
	// PID for instrument joint position
	m_instruJntCtrl:ARRAY[1..5] OF FB_PID;

	// PID for instrument yaw angle 
	m_instruYawCtrl : FB_PID;
	
	// command instrument joint position and velocity
	m_instruCmdJntPos:Vec5d;
	m_instruCmdJntVel:Vec5d;
	
	// current instrument joint position and velocity
	m_instruCurJntPos: Vec5d;
	m_instruCurJntVel:Vec5d;
	
	// grasp force level
	m_graspForceLevel:Lreal :=0;
	
	// instrument joint control torque(when gripper is open)
	m_instruJntCtrlTrq:Vec5d:=[5(0.0)];

	// instrument yaw control torque(when gripper is closed)
	m_instruYawCtrlTrq:LREAL;
		
	// current gripper yaw velocity
	m_instruCurYawVel:LREAL;
	
	// yaw angle error(deg)
	m_yawAngErr : LREAL;
	
	// backlash compensation variables
	m_jntBacklash:ARRAY[1..5] OF LREAL:=[5(0)];
	m_instruLastCmdJntPos:Vec5d;
	
	// grip yaw compensation variables
 	m_gripYawCompAng :LREAL;
 	m_maxGripYawCompAng :LREAL;
	m_lastCmdYawAng:LREAL;
	m_jntMoveStep:LREAL := 0.5*g_deg2Rad;
	
END_VAR

METHOD calcBacklash : BOOL
VAR_IN_OUT CONSTANT
	// instrument joint command position
	i_cmdInstruJntPos :Vec5d;
	
	// command yaw position
	i_cmdYawPos : LREAL;
	
	// slave arm data
	i_slaveArm :FB_SlaveArm;
END_VAR

VAR
	i:INT;
	deltaAng:LREAL;
END_VAR
// backslash compensation
FOR i:=1 TO 4 DO
	// integral compensated backslash angle
	deltaAng:=i_cmdInstruJntPos[i]-m_instruLastCmdJntPos[i];
	IF ABS(deltaAng)>m_jntMoveStep THEN
		m_jntBacklash [i] := m_jntBacklash [i] + m_jntMoveStep*sign(deltaAng);
		m_instruLastCmdJntPos[i] := i_cmdInstruJntPos[i];
	END_IF
END_FOR


// exert grip force 
IF m_graspForceLevel >0  THEN
	
	// clear grip finger backlash
	m_jntBacklash [1]:=0;
	m_jntBacklash [2]:=0;
	
	// determin max compensated angle based on grip force 
	FOR i:=1 TO 4 DO 
		IF m_graspForceLevel<= g_instruGripYawCompForceLevel[i] THEN
			m_maxGripYawCompAng := g_instruGripYawCompAng[i];
			EXIT;
		END_IF
	END_FOR

	// compensate yaw joint angle in case it's driven by force difference between two fingers
	IF m_graspForceLevel > 80 AND  ABS(i_cmdYawPos - m_lastCmdYawAng) > m_jntMoveStep  THEN
		m_jntBacklash [3] := m_jntBacklash [3] -  4*m_jntMoveStep*sign(i_cmdYawPos - m_lastCmdYawAng);
	END_IF
	
	// determin  compensated angle
	IF ABS(i_cmdYawPos - m_lastCmdYawAng) > m_jntMoveStep  THEN
		// determin  compensated yaw  angle
		IF (i_cmdYawPos - m_lastCmdYawAng) * m_gripYawCompAng <= 0 THEN
			m_gripYawCompAng := m_gripYawCompAng + 4*m_jntMoveStep * sign(i_cmdYawPos-m_lastCmdYawAng);
		ELSE
			m_gripYawCompAng := m_gripYawCompAng + 2*m_jntMoveStep * sign(i_cmdYawPos-m_lastCmdYawAng);
		END_IF
		m_lastCmdYawAng := i_cmdYawPos;
	END_IF
	m_gripYawCompAng := LIMIT(-m_maxGripYawCompAng, m_gripYawCompAng,m_maxGripYawCompAng);
	

ELSE
	m_gripYawCompAng:=0;
	m_lastCmdYawAng := i_cmdYawPos;
END_IF

// limit compensated backslash angle
FOR i:=1 TO 4 DO

	IF i<3 THEN 
		IF g_instruBacklashDir[i] > 0 THEN
			m_jntBacklash [i] := LIMIT(0, m_jntBacklash[i], i_slaveArm.instrument.instruTypeInfo.m_instruYawBacklash);		
		ELSE
			m_jntBacklash [i] := LIMIT(-i_slaveArm.instrument.instruTypeInfo.m_instruYawBacklash, m_jntBacklash[i], 0);	
		END_IF

	ELSIF i=3 THEN
		IF g_instruBacklashDir[i] > 0 THEN
			m_jntBacklash [i] := LIMIT(0, m_jntBacklash[i], i_slaveArm.instrument.instruTypeInfo.m_instruPitchBachlash);
		ELSE
			m_jntBacklash [i] := LIMIT(-i_slaveArm.instrument.instruTypeInfo.m_instruPitchBachlash, m_jntBacklash[i], 0);	
		END_IF
	ELSE
		m_jntBacklash [i]:=0;
	END_IF
	
END_FOR
END_METHOD

METHOD PUBLIC clearBacklash : BOOL
VAR_INPUT
END_VAR
m_jntBacklash := g_zeroVec5d;
END_METHOD

METHOD init : BOOL
VAR_IN_OUT CONSTANT
	i_slaveArm:FB_SlaveArm;
END_VAR

VAR
	i,j:INT;
END_VAR
m_graspForceLevel:=0;

// init controller
m_maxGripCurrent:= i_slaveArm.instrument.instruTypeInfo.m_normGripTrq;
m_currentRatioMotor2Jnt:=GVL_SlaveMotorParameters.g_motorTrqConst[4]*GVL_SlaveMotorParameters.g_motorReduction[4]/1000;
m_maxGripForce := m_maxGripCurrent * m_currentRatioMotor2Jnt;
m_maxGripCtrlForce := m_maxGripCtrlCurrent * m_currentRatioMotor2Jnt;
FOR i:=1 TO 4 DO
	m_instruCmdJntPos[i]:=i_slaveArm.curJntPos[i+3];
	
	m_instruCmdJntVel[i]:=0;
	
	m_instruJntCtrl[i].init(g_slaveArmCtrlCycleTime,m_instruKp[i],m_instruKd[i],m_instruKi[i],
		m_instruKiLimit[i]* m_currentRatioMotor2Jnt,	m_instruCtrlLimit[i]*m_currentRatioMotor2Jnt);
	
	m_instruLastCmdJntPos[i]:=m_instruCmdJntPos[i];
END_FOR
m_instruYawCtrl.init(g_slaveArmCtrlCycleTime,m_yawKp[1],m_yawKd[1],m_yawKi[1],m_yawKiLimit*m_currentRatioMotor2Jnt, m_yawCtrlLimit*m_currentRatioMotor2Jnt);
END_METHOD

METHOD run : BOOL
VAR_IN_OUT CONSTANT
	// instrument joint command position
	i_cmdInstruJntPos :Vec5d;
	
	// instrument joint command velocity
	i_cmdInstruJntVel :Vec5d;
	
	// command yaw position
	i_cmdYawPos : LREAL;
	
	// command yaw velocity
	i_cmdYawVel :LREAL;
	
	// command grip force level
	i_cmdGripForceLevel:LREAL;
	
	// slave arm data
	i_slaveArm :FB_SlaveArm;
END_VAR

VAR_OUTPUT
	// joint control torque
	o_cmdJntTrq:Vec5d;
END_VAR

VAR
	i: INT;
	deltaAng:LREAL;
END_VAR
m_graspForceLevel:=LIMIT(0,i_cmdGripForceLevel ,  100)	;

// calculate instrument backlash
calcBacklash(i_cmdInstruJntPos, i_cmdYawPos, i_slaveArm);


// joint position control
FOR i:=1 TO 4 DO	
	m_instruCmdJntPos[i]:=i_cmdInstruJntPos[i];
	m_instruCmdJntVel[i]:=i_cmdInstruJntVel[i];
	m_instruCurJntPos[i]:=i_slaveArm.curJntPos[i+3];
	m_instruCurJntVel[i]:= i_slaveArm.curJntVel[i+3];
	m_instruJntCtrlTrq[i]:=m_instruJntCtrl[i].run(m_instruCmdJntPos[i] ,m_instruCurJntPos[i], m_instruCmdJntVel[i], m_instruCurJntVel[i]);
END_FOR
m_instruJntCtrlTrq[5]:=0;

m_instruCurYawVel :=i_slaveArm.curDHJntVel[6];
m_yawAngErr:=g_rad2Deg*(i_cmdYawPos-i_slaveArm.curDHJntPos[6]);


// exert grip force 
IF m_graspForceLevel >0  THEN
	
	// varialbe PID control based on different gripper force level
	FOR i:=1 TO 3 DO 
		IF m_graspForceLevel < m_forceLevelThres[i] THEN
			m_instruYawCtrl.setPIDParam(m_yawKp[i],m_yawKd[i],m_yawKi[i]);
			EXIT;
		END_IF
	END_FOR

	// yaw control
	m_instruYawCtrlTrq:=m_instruYawCtrl.run(i_cmdYawPos+m_gripYawCompAng,i_slaveArm.curDHJntPos[6],i_cmdYawVel, m_instruCurYawVel);

	// add feed forward grasp force
	m_instruJntCtrlTrq[1]:= m_maxGripForce*m_graspForceLevel/100.0 + m_instruYawCtrlTrq;
	m_instruJntCtrlTrq[2]:= m_maxGripForce*m_graspForceLevel/100.0 - m_instruYawCtrlTrq;
	m_instruJntCtrlTrq[1]:=LIMIT(-m_maxGripForce/10.0,m_instruJntCtrlTrq[1], m_maxGripCtrlForce);
	m_instruJntCtrlTrq[2]:=LIMIT(-m_maxGripForce/10.0,m_instruJntCtrlTrq[2], m_maxGripCtrlForce);
END_IF

o_cmdJntTrq := m_instruJntCtrlTrq;
END_METHOD

METHOD setMaxGripTrq : BOOL
VAR_INPUT
	i_maxGripTrq:LREAL;
END_VAR
m_maxGripCurrent := i_maxGripTrq;
m_maxGripForce := m_maxGripCurrent * m_currentRatioMotor2Jnt;
END_METHOD

END_FUNCTION_BLOCK

// ---- FBs_BasicControllers/FB_UltrosonicKnifeControl.TcPOU
// instrument joints control
FUNCTION_BLOCK FB_UltrosonicKnifeControl
VAR_INPUT
END_VAR
VAR_OUTPUT
END_VAR
VAR
	// instrument PID control paramters
	m_instruKp:ARRAY[1..5] OF LREAL:=[5(5)];
	m_instruKd:ARRAY[1..5] OF LREAL:=[5(0.25)];
	m_instruKi:ARRAY[1..5] OF LREAL:=[5(10.0)];
	m_instruKiLimit:ARRAY[1..5] OF LREAL:=[5(50.0)];
	m_instruCtrlLimit:ARRAY[1..5] OF LREAL:=[4(150.0), 200.0];
	
	// max grip force/current(mA)
	m_maxGripForce:LREAL;
	m_maxGripCurrent:LREAL:=150.0;
	
	// PID for instrument joint position
	m_instruJntCtrl:ARRAY[1..5] OF FB_PID;
	
	// ratio convert motor current to joint troque
	m_currentRatioMotor2Jnt:LREAL;

	// command instrument joint position and velocity
	m_instruCmdJntPos:Vec5d;
	m_instruLastCmdJntPos:Vec5d;
	m_instruCmdJntVel:Vec5d;
	
	// backlash compensation variables
	m_jntBacklash:ARRAY[1..5] OF LREAL:=[5(0)];
	m_jntMoveStep:LREAL := 0.5*g_deg2Rad;
	
	// current instrument joint position and velocity
	m_instruCurJntPos: Vec5d;
	m_instruCurJntVel:Vec5d;
	
	// grasp force level
	m_graspForceLevel:Lreal :=0;
	
	// instrument joint control torque(when gripper is open)
	m_instruJntCtrlTrq:Vec5d:=[5(0.0)];
	
	// minimum grip angle to apply grip force; convert grasp force level to minus grip angle
	m_minGripAngle :LREAL := -60*g_deg2Rad;
	m_gripForceAngle:LREAL;

END_VAR

METHOD calcBacklash : BOOL
VAR_IN_OUT CONSTANT
	// instrument joint command position
	i_cmdInstruJntPos :Vec5d;
	
	// slave arm data
	i_slaveArm :FB_SlaveArm;
END_VAR

VAR
	i:INT;
	deltaAng:LREAL;
END_VAR
// backslash compensation
FOR i:=3 TO 3 DO
	// integral compensated backslash angle
	deltaAng:=i_cmdInstruJntPos[i]-m_instruLastCmdJntPos[i];
	IF ABS(deltaAng)>m_jntMoveStep THEN
		m_jntBacklash [i] := m_jntBacklash [i] + m_jntMoveStep*sign(deltaAng);
		m_instruLastCmdJntPos[i] := i_cmdInstruJntPos[i];
	END_IF
END_FOR


// exert grip force 
IF m_graspForceLevel >0  THEN
	
	// max grip finger backlash
	m_jntBacklash [3]:=-i_slaveArm.instrument.instruTypeInfo.m_instruYawBacklash;
	
END_IF

// limit compensated backslash angle
FOR i:=3 TO 3 DO
	IF g_instruBacklashDir[i] > 0 THEN
		m_jntBacklash [i] := LIMIT(0, m_jntBacklash[i], i_slaveArm.instrument.instruTypeInfo.m_instruYawBacklash);
	ELSE
		m_jntBacklash [i] := LIMIT(-i_slaveArm.instrument.instruTypeInfo.m_instruYawBacklash, m_jntBacklash[i], 0);	
	END_IF
	
END_FOR
END_METHOD

METHOD PUBLIC clearBacklash : BOOL
VAR_INPUT
END_VAR
m_jntBacklash := g_zeroVec5d;
END_METHOD

METHOD init : BOOL
VAR_IN_OUT CONSTANT
	i_slaveArm:FB_SlaveArm;
END_VAR

VAR
	i,j:INT;
END_VAR
m_graspForceLevel:=0;

// init controller
m_instruCtrlLimit[3] := i_slaveArm.instrument.instruTypeInfo.m_normGripTrq;
m_currentRatioMotor2Jnt:=GVL_SlaveMotorParameters.g_motorTrqConst[4]*GVL_SlaveMotorParameters.g_motorReduction[4]/1000;
m_maxGripForce := m_maxGripCurrent * m_currentRatioMotor2Jnt;
FOR i:=1 TO 5 DO
	m_instruCmdJntPos[i]:=i_slaveArm.curJntPos[i+3];
	m_instruLastCmdJntPos[i]:=m_instruCmdJntPos[i];
	m_instruCmdJntVel[i]:=0;
	
	m_instruJntCtrl[i].init(g_slaveArmCtrlCycleTime,m_instruKp[i],m_instruKd[i],m_instruKi[i],
		m_instruKiLimit[i]* m_currentRatioMotor2Jnt,	m_instruCtrlLimit[i]*m_currentRatioMotor2Jnt);
END_FOR
END_METHOD

METHOD run : BOOL
VAR_IN_OUT CONSTANT
	// instrument joint command position
	i_cmdInstruJntPos :Vec5d;
	
	// instrument joint command velocity
	i_cmdInstruJntVel :Vec5d;
	
	// command grip force level
	i_cmdGripForceLevel:LREAL;
	
	// slave arm data
	i_slaveArm :FB_SlaveArm;
END_VAR

VAR_OUTPUT
	// joint control torque
	o_cmdJntTrq:Vec5d;
END_VAR

VAR
	i: INT;
END_VAR
// calculate instrument backlash
calcBacklash(i_cmdInstruJntPos, i_slaveArm);

// convert force level to grip angle
m_graspForceLevel:=LIMIT(0,i_cmdGripForceLevel , 100);
m_gripForceAngle:=m_minGripAngle*m_graspForceLevel/100;

// joint position control
FOR i:=1 TO 5 DO	
	m_instruCmdJntPos[i]:=i_cmdInstruJntPos[i];
	m_instruCmdJntVel[i]:=i_cmdInstruJntVel[i];
	m_instruCurJntPos[i]:=i_slaveArm.curJntPos[i+3];
	m_instruCurJntVel[i]:= i_slaveArm.curJntVel[i+3];
	IF i=3 THEN
		m_instruCmdJntPos[i]:=i_cmdInstruJntPos[i]+m_gripForceAngle;
	END_IF
	m_instruJntCtrlTrq[i]:=m_instruJntCtrl[i].run(m_instruCmdJntPos[i],m_instruCurJntPos[i], m_instruCmdJntVel[i], m_instruCurJntVel[i]);
END_FOR
m_instruJntCtrlTrq[1]:=0;
m_instruJntCtrlTrq[2]:=0;
m_instruJntCtrlTrq[4]:=0;

// exert grip force 
//IF m_graspForceLevel >0  THEN
//	m_instruJntCtrlTrq[3]:= -m_maxGripForce*m_graspForceLevel/100.0;	
//END_IF

o_cmdJntTrq := m_instruJntCtrlTrq;
END_METHOD

END_FUNCTION_BLOCK

// ---- AgiMaths/MatrixLib/angAxis2Rot.TcPOU
FUNCTION angAxis2Rot : Mat3d
VAR_INPUT
	i_angle :LREAL;
	i_axis :Vec3d;
END_VAR
VAR
	cAng, sAng :LREAL;
	rx,ry,rz :LREAL;
END_VAR

IF norm(i_axis)<g_smallNum THEN
	angAxis2Rot := g_eye3d;
	RETURN;
END_IF

cAng :=COS(i_angle);
sAng := SIN(i_angle);
rx:=i_axis[1];
ry:=i_axis[2];
rz:=i_axis[3];

angAxis2Rot[1,1]:=rx*rx*(1-cAng)+cAng;
angAxis2Rot[2,1]:=rx*ry*(1-cAng)+rz*sAng;
angAxis2Rot[3,1]:=rx*rz*(1-cAng)-ry*sAng;

angAxis2Rot[1,2]:=rx*ry*(1-cAng)-rz*sAng;
angAxis2Rot[2,2]:=ry*ry*(1-cAng)+cAng;
angAxis2Rot[3,2]:=ry*rz*(1-cAng)+rx*sAng;

angAxis2Rot[1,3]:=rx*rz*(1-cAng)+ry*sAng;
angAxis2Rot[2,3]:=ry*rz*(1-cAng)-rx*sAng;
angAxis2Rot[3,3]:=rz*rz*(1-cAng)+cAng;

END_FUNCTION

// ---- AgiMaths/MatrixLib/vecSelfAdd.TcPOU
// A +=B
FUNCTION vecSelfAdd : BOOL
VAR_IN_OUT
	vecA :ARRAY[*] OF LREAL;
END_VAR

VAR_IN_OUT CONSTANT
	vecB :ARRAY[*] OF LREAL;
END_VAR

VAR
	m,i :DINT;
 
END_VAR

m:=UPPER_BOUND(vecA,1);

FOR i:=1 TO m DO
		vecA[i]:=vecA[i]+vecB[i];
END_FOR

END_FUNCTION

// ---- AgiMaths/MatrixLib/invMat2.TcPOU
FUNCTION invMat2 : bool
VAR_IN_OUT CONSTANT
	mat :Mat2d;
END_VAR
VAR_IN_OUT
	invMat : Mat2d;
END_VAR
VAR
	matDet:LREAL;
END_VAR

matDet := mat[1,1]*mat[2,2]-mat[1,2]*mat[2,1];

IF ABS(matDet)<g_smallNum THEN
	invMat2 := FALSE;
	RETURN;
END_IF

invMat[1,1]:= mat[2,2]/matDet;
invMat[1,2]:= -mat[1,2]/matDet;
invMat[2,1]:= -mat[2,1]/matDet;
invMat[2,2]:= mat[1,1]/matDet;
 
invMat2:=TRUE;

END_FUNCTION

// ---- FBs_SlaveControllers/FB_SlaveCtrlScopeReady.TcPOU
// Brief:Scope Ready
FUNCTION_BLOCK PUBLIC FB_SlaveCtrlScopeReady EXTENDS FB_SlaveArmCtrlBase
VAR_INPUT
END_VAR
VAR_OUTPUT
END_VAR
VAR
END_VAR

METHOD PUBLIC init : BOOL
VAR_IN_OUT CONSTANT
	i_slaveArm	:FB_SlaveArm;
END_VAR
VAR_IN_OUT 
	r_slaveArmCtrlCmd :ST_SlaveArmCtrlCmds;
END_VAR


VAR
	j:INT;
	maxJntErr:LREAL;
	jntCtrlErr:Vec7d;
END_VAR
// check if to hold the command joint position unchanged
m_holdLastCmds := checkToHoldLastCmds(i_slaveArm);

//init
SUPER^.Init(i_slaveArm,r_slaveArmCtrlCmd);
END_METHOD

END_FUNCTION_BLOCK

// ---- FBs_SlaveControllers/FB_SlaveCtrlEndoscope.TcPOU
// Brief: Slave Arm Endoscope Control
FUNCTION_BLOCK PUBLIC FB_SlaveCtrlEndoscope EXTENDS FB_SlaveArmCtrlBase
VAR_INPUT
END_VAR
VAR_OUTPUT
END_VAR
VAR
	// scope motion master-salve scale
	m_MSMotionScale :LREAL :=-0.3;
	
	// scope motion singularity scale
	m_singMotionScale :LREAL :=1;
	m_minSingMotionScale :LREAL := 0.4;
	
	// distance threshold between scope and remote center without sigularity scale 
	m_RCDisThres :LREAL :=0.1;
	
	// filter cut-off frequency for master-slave control
	m_cmdJntPosLpfCutoffFreq : LREAL :=5;
	
	// last command joint position
	m_lastCmdJntPos :Vec8d;
	
	// command velocity filter
	m_cmdVelLpf:ARRAY[1..4] OF FB_LowPassFilter;
	
	// scope command linear/rotate velocity in local/view coordinate
	m_cmdVelLocal :Vec3d;
	m_cmdWVelLocal :LREAL;
	
	// scope command linear velocity in base coordinate
	m_cmdVel:Vec3d;
	
	// rotate compensation velocity 
	m_rotCompVel :LREAL;
	
END_VAR

METHOD PROTECTED calcCmdJntPos : BOOL
VAR_IN_OUT CONSTANT
	i_endoscopePose : ST_Frame;
	i_masterStatus :ST_MasterStatus;
	i_setupStatus: ST_SetupStatus;
	i_slaveArm :FB_SlaveArm;
END_VAR

VAR 
	i,j : INT;
	posJaco, posJacoInv:Mat3d;
	armDHJntVel :Vec3d;

	cmdVelScale :LREAL;
	jnt3Limit :LREAL;
	scopeRotJntIdx:INT:=8;
END_VAR
IF isFinished THEN
	RETURN;
END_IF

// compute desired view velocity
cmdVelCalc(i_masterStatus, i_slaveArm);

// filt command velocity
m_cmdVelLocal[1] := m_cmdVelLpf[1].run(m_cmdVelLocal[1]);
m_cmdVelLocal[2] := m_cmdVelLpf[2].run(m_cmdVelLocal[2]);
m_cmdVelLocal[3] := m_cmdVelLpf[3].run(m_cmdVelLocal[3]);
m_cmdWVelLocal := -m_cmdVelLpf[4].run(m_cmdWVelLocal);

// get linear velocity in base
matMultiVec(i_slaveArm.simCartPose.m_rot, m_cmdVelLocal, m_cmdVel);

// position jacobian and its inverse
FOR i:=1 TO 3 DO
	FOR j:=1 TO 3 DO
		posJaco[i,j]:=i_slaveArm.simJaco[i,j];
	END_FOR 
END_FOR
invMat3(posJaco, posJacoInv);

// command joint velocity of joint 1-3
matMultiVec(posJacoInv, m_cmdVel, armDHJntVel);

// limit DH joints velocity 
cmdVelScale := 1;
FOR i:=1 TO 3 DO 
	cmdVelScale:=MAX(cmdVelScale, ABS(armDHJntVel[i]/GVL_SlaveMotorParameters.g_maxJntVel[i]));
END_FOR
vecSelfMultiNum(armDHJntVel, 1.0/cmdVelScale);

// limit arm joint position
FOR i:=1 TO 3 DO
	IF (armDHJntVel[i] > 0 AND  i_slaveArm.simDHJntPos[i] + armDHJntVel[i]*g_slaveArmCtrlCycleTime> GVL_SlaveMotorParameters.g_maxDHJntPos[i]) OR 
		(armDHJntVel[i] <0 AND	i_slaveArm.simDHJntPos[i] + armDHJntVel[i]*g_slaveArmCtrlCycleTime< GVL_SlaveMotorParameters.g_minDHJntPos[i]) THEN
		armDHJntVel[i]:=0;
	END_IF
END_FOR

// joint 3 up limit to remote center
jnt3Limit := i_slaveArm.instrument.instruTypeInfo.m_rodLength - GVL_SlaveArmKinematic.g_minInstruRCDis;
IF (armDHJntVel[3] > 0 AND  i_slaveArm.simDHJntPos[3] + armDHJntVel[3]*g_slaveArmCtrlCycleTime> jnt3Limit) THEN
	armDHJntVel[3]:=0;
END_IF

// final arm joint command velocity
m_cmdJntVel[1]:= armDHJntVel[1];
m_cmdJntVel[2]:= armDHJntVel[2];
m_cmdJntVel[3]:= armDHJntVel[3];

// limit rotate joint veloicyt
m_cmdWVelLocal := LIMIT (-GVL_SlaveMotorParameters.g_maxJntVel[8],  m_cmdWVelLocal, GVL_SlaveMotorParameters.g_maxJntVel[8]);

// as there are two types scope holder, need to determin the rotate joint index
IF i_slaveArm.instrument.onChipData.m_InstruID = InstruType_NewEndoscope THEN
	scopeRotJntIdx :=7;
	m_jntOPMode[6] := DriverOPMode_Trq;
ELSE
	scopeRotJntIdx:=8;
END_IF

// compensate view rotation cause by joint6 
m_rotCompVel := rotateCompensate(i_slaveArm);

m_cmdJntVel[scopeRotJntIdx]:= (m_rotCompVel-m_cmdWVelLocal)/i_slaveArm.instrument.m_endoscopeRotateReduction;

// integral to command joint position
m_cmdJntPos[1]:=m_simJntPos[1]+m_cmdJntVel[1]*g_slaveArmCtrlCycleTime;
m_cmdJntPos[2]:=m_simJntPos[2]+m_cmdJntVel[2]*g_slaveArmCtrlCycleTime;
m_cmdJntPos[3]:=m_simJntPos[3]+m_cmdJntVel[3]*g_slaveArmCtrlCycleTime;
m_cmdJntPos[scopeRotJntIdx]:=m_simJntPos[scopeRotJntIdx]+m_cmdJntVel[scopeRotJntIdx]*g_slaveArmCtrlCycleTime;

// joint6 output torque to help rotation motion
IF m_jntOPMode[6] = DriverOPMode_Trq THEN
	m_cmdJntTrq[6] := -0.5*i_slaveArm.cmdJntTrq[7];
END_IF


m_simJntPos := m_cmdJntPos;
END_METHOD

METHOD PROTECTED cmdVelCalc : BOOL
VAR_IN_OUT CONSTANT
	i_masterStatus :ST_MasterStatus;
	i_slaveArm :FB_SlaveArm;
END_VAR

VAR
	leftVel, rightVel :Vec3d;
	i:INT;
	radiusVec :Vec3d;
	radiusLength :LREAL;
	leftWVel, rightWVel :Vec3d;
END_VAR
FOR i :=1 TO 3 DO 
	leftVel[i] := i_masterStatus.m_curArmTwist[1][i];
	rightVel[i] := i_masterStatus.m_curArmTwist[2][i];
END_FOR

// master linear velocity
vecAdd(leftVel, rightVel , m_cmdVelLocal);
vecSelfMultiNum(m_cmdVelLocal, 0.5);

// motion scale
//m_singMotionScale := motionScale(i_slaveArm); // NOTE: velocity scale near singularity is disable current
vecSelfMultiNum(m_cmdVelLocal, m_MSMotionScale);

// radius vector from right arm to left arm
vecSub(i_masterStatus.m_curArmPose[1].m_pos, i_masterStatus.m_curArmPose[2].m_pos, radiusVec);
vecSelfMultiNum(radiusVec, 0.5);
radiusVec[3]:=0;
radiusLength := norm(radiusVec);
normalize(radiusVec);

// left rotate velocity
leftVel[3]:= 0;
leftWVel := cross(radiusVec, leftVel);

// right rotate velocity
// radius vector from left arm to right arm
vecSelfMultiNum(radiusVec, -1.0);
rightVel[3]:= 0;
rightWVel := cross(radiusVec, rightVel);

m_cmdWVelLocal:= (leftWVel[3] + rightWVel[3])/(2.0*radiusLength);
END_METHOD

METHOD PUBLIC init : BOOL
VAR_IN_OUT CONSTANT
	i_slaveArm	:FB_SlaveArm;
END_VAR
VAR_IN_OUT 
	r_slaveArmCtrlCmd :ST_SlaveArmCtrlCmds;
END_VAR
VAR 
	i :INT ;
END_VAR
SUPER^.Init(i_slaveArm,r_slaveArmCtrlCmd);
m_simJntPos :=m_cmdJntPos;
m_lastCmdJntPos :=m_cmdJntPos;
m_jntOPMode := g_slaveAllPosTrqMode;

// init filter
FOR i:=1 TO 4 DO
	m_cmdVelLpf[i].init(1, m_cmdJntPosLpfCutoffFreq, g_slaveArmCtrlFreq);
END_FOR

// update commands to arm
copyCmds(r_slaveArmCtrlCmd);
END_METHOD

METHOD PROTECTED motionScale : LREAL
VAR_IN_OUT CONSTANT
	i_slaveArm :FB_SlaveArm;
END_VAR
VAR
	RCDis :LREAL;
END_VAR
RCDis := ABS(i_slaveArm.curJntPos[3] - i_slaveArm.instrument.instruTypeInfo.m_rodLength);

IF RCDis < GVL_SlaveArmKinematic.g_minInstruRCDis THEN
	motionScale := m_minSingMotionScale;
ELSIF RCDis > m_RCDisThres THEN
	motionScale :=1 ;
ELSE
	motionScale := m_minSingMotionScale + (1- m_minSingMotionScale) * (RCDis - GVL_SlaveArmKinematic.g_minInstruRCDis)/(m_RCDisThres - GVL_SlaveArmKinematic.g_minInstruRCDis);
	motionScale := LIMIT(0, motionScale, 1.0);
END_IF
END_METHOD

METHOD rotateCompensate : LREAL
VAR_IN_OUT CONSTANT
	i_slaveArm :FB_SlaveArm;
END_VAR
VAR
	rotJaco:Mat3d;
	armJntVel:Vec3d;
	i,j:INT;
	wVelWrd :Vec3d;
	jnt4JacoInv :Vec3d;
	jnt4JacoNorm:LREAL;
	rotT:Mat3d;
END_VAR
FOR i:=1 TO 3 DO 
	FOR j:=1 TO 3 DO 
		rotJaco[i,j] := i_slaveArm.jaco[i+3, j];
	END_FOR
	armJntVel[i] := m_cmdJntVel[i];
	jnt4JacoInv[i] := i_slaveArm.jaco[i+3,4];
END_FOR

// get rotate velocity 
MatMultiVec(rotJaco, armJntVel, wVelWrd);

jnt4JacoNorm := norm(jnt4JacoInv);
vecSelfMultiNum(jnt4JacoInv, 1.0/(jnt4JacoNorm*jnt4JacoNorm));

rotateCompensate := -vecDot(jnt4JacoInv, wVelWrd);
END_METHOD

END_FUNCTION_BLOCK

// ---- FBs_SlaveControllers/FB_SlaveCtrlAdjust.TcPOU
// Brief: Slave Arm Adjust
FUNCTION_BLOCK PUBLIC FB_SlaveCtrlAdjust EXTENDS FB_SlaveArmCtrlBase
VAR
	// velocity for full damping
	m_maxAdjustVel :Vec3d := [1.2, 1.2, 0.3];
	
	// velocity start to enable damping
	m_velLBForDamp :Vec3d := [1.0, 1.0, 0.2];
	
	// max damp
	m_maxDamp :Vec3d := [50, 50, 500];
	
	// distance buffer from joint limit to start damp
	m_limitBufferForDamp :Vec3d :=[20*g_deg2Rad, 20*g_deg2Rad, 0.03];
	
END_VAR

// override this function in each exact controller
METHOD PROTECTED calcCmdJntPos : BOOL
VAR_IN_OUT CONSTANT
	i_endoscopePose : ST_Frame;
	i_masterStatus :ST_MasterStatus;
	i_setupStatus: ST_SetupStatus;
	i_slaveArm :FB_SlaveArm;
END_VAR
m_cmdJntPos[1]:=i_slaveArm.curJntPos[1];
m_cmdJntPos[2]:=i_slaveArm.curJntPos[2];
m_cmdJntPos[3]:=i_slaveArm.curJntPos[3];
IF m_jntOPMode[8] = DriverOPMode_Trq THEN
	m_cmdJntPos[8]:=i_slaveArm.curJntPos[8];
END_IF
IF m_jntOPMode[7] = DriverOPMode_Trq THEN
	m_cmdJntPos[7]:=i_slaveArm.curJntPos[7];
END_IF

m_cmdCartPose:=i_slaveArm.curCartPose;
END_METHOD

// override this function in each exact controller
METHOD PROTECTED calcCmdJntTrq : BOOL
VAR_IN_OUT CONSTANT
	i_endoscopePose : ST_Frame;
	i_masterStatus :ST_MasterStatus;
	i_setupStatus: ST_SetupStatus;
	i_slaveArm :FB_SlaveArm;
END_VAR
VAR
	i :INT;
	dampScale :LREAL;
	limitDis:LREAL;
END_VAR
// set joint torque to zero in default
m_cmdJntTrq := g_zeroVec8d;

// enable endoscope rotation joint if external torque exceed specific value
IF i_slaveArm.instrument.onChipData.m_InstruReadSucceed AND i_slaveArm.instrument.instruType = InstruType_Endoscope AND ABS(i_slaveArm.filtJntCurrent[8]) > 100 THEN
		m_jntOPMode[8]:=DriverOPMode_Trq;
END_IF


// add damp near joint limit
FOR i:=1 TO 3 DO
	IF (i_slaveArm.curJntPos[i] > GVL_SlaveMotorParameters.g_maxDHJntPos[i] - m_limitBufferForDamp[i] AND  i_slaveArm.curJntVel[i]> 0 ) 
		OR (i_slaveArm.curJntPos[i] < GVL_SlaveMotorParameters.g_minDHJntPos[i] + m_limitBufferForDamp[i] AND  i_slaveArm.curJntVel[i]<0 )  THEN
		limitDis := MIN(GVL_SlaveMotorParameters.g_maxDHJntPos[i] - i_slaveArm.curJntPos[i], i_slaveArm.curJntPos[i]-GVL_SlaveMotorParameters.g_minDHJntPos[i]);
		dampScale  :=LIMIT(0, 1-limitDis/m_limitBufferForDamp[i],1);
		m_cmdJntTrq[i]:= -dampScale * m_maxDamp[i] * i_slaveArm.curJntVel[i];
	END_IF
	
END_FOR

// compute damp
FOR i:=1 TO 3 DO
	IF ABS(i_slaveArm.curJntVel[i]) > m_velLBForDamp[i] THEN 
		dampScale:=LIMIT(0, (ABS(i_slaveArm.curJntVel[i])- m_velLBForDamp[i])/(m_maxAdjustVel[i] - m_velLBForDamp[i]), 1 );
		m_cmdJntTrq[i] :=m_cmdJntTrq[i] -i_slaveArm.curJntVel[i] * m_maxDamp[i] * dampScale;
	END_IF
END_FOR
END_METHOD

METHOD PUBLIC init : BOOL
VAR_IN_OUT CONSTANT
	i_slaveArm	:FB_SlaveArm;
END_VAR
VAR_IN_OUT 
	r_slaveArmCtrlCmd :ST_SlaveArmCtrlCmds;
END_VAR
VAR
	i :INT;
END_VAR
// check if to hold the command joint position unchanged
m_holdLastCmds := checkToHoldLastCmds(i_slaveArm);

//init
SUPER^.Init(i_slaveArm,r_slaveArmCtrlCmd);

// disable joints if this joint is an unrecoverable failure
FOR i:=1 TO g_sJntNum DO
	IF SafetyCheck.m_SafetyCheck.m_jntErrFlag[i_slaveArm.armIdx, 0, 3] OR  SafetyCheck.m_SafetyCheck.m_jntErrFlag[i_slaveArm.armIdx, i+g_setupJntNum, 3] THEN
		m_jntEnableFlag[i] := 0;
	ELSE
		m_jntEnableFlag[i] := 1;
	END_IF
END_FOR

// joint 1/2/3/7 run in torque mode
m_jntOPMode[1]:=DriverOPMode_Trq;
m_jntOPMode[2]:=DriverOPMode_Trq;
m_jntOPMode[3]:=DriverOPMode_Trq;
m_jntOPMode[4]:=DriverOPMode_PosTrq;
m_jntOPMode[5]:=DriverOPMode_PosTrq;
m_jntOPMode[6]:=DriverOPMode_PosTrq;
m_jntOPMode[7]:=DriverOPMode_PosTrq;
m_jntOPMode[8]:=DriverOPMode_PosTrq;

IF i_slaveArm.instrument.onChipData.m_InstruReadSucceed THEN
	IF i_slaveArm.instrument.instruType <> InstruType_Endoscope THEN
		m_jntOPMode[7]:=DriverOPMode_Trq;
	END_IF
END_IF

// update commands to arm
copyCmds(r_slaveArmCtrlCmd);
END_METHOD

END_FUNCTION_BLOCK

// ---- FBs_SlaveControllers/FB_SlaveCtrlPackage.TcPOU
// Brief: Slave Arm move to Package posture
FUNCTION_BLOCK PUBLIC FB_SlaveCtrlPackage EXTENDS FB_SlaveArmCtrlBase
VAR_INPUT
END_VAR
VAR_OUTPUT
END_VAR
VAR
END_VAR

METHOD PUBLIC init : BOOL
VAR_IN_OUT CONSTANT
	i_slaveArm	:FB_SlaveArm;
END_VAR
VAR_IN_OUT 
	r_slaveArmCtrlCmd :ST_SlaveArmCtrlCmds;
END_VAR
// check if to hold the command joint position unchanged
m_holdLastCmds := checkToHoldLastCmds(i_slaveArm);

//init
SUPER^.Init(i_slaveArm,r_slaveArmCtrlCmd);
END_METHOD

END_FUNCTION_BLOCK

// ---- FBs_SlaveControllers/FB_SlaveCtrlCart.TcPOU
// Brief: Slave Arm Cart Control
FUNCTION_BLOCK PUBLIC FB_SlaveCtrlCart EXTENDS FB_SlaveArmCtrlBase
VAR_INPUT
END_VAR
VAR_OUTPUT
END_VAR
VAR
END_VAR

METHOD PUBLIC init : BOOL
VAR_IN_OUT CONSTANT
	i_slaveArm	:FB_SlaveArm;
END_VAR
VAR_IN_OUT 
	r_slaveArmCtrlCmd :ST_SlaveArmCtrlCmds;
END_VAR

VAR
	j:INT;
	maxJntErr:LREAL;
	jntCtrlErr:Vec7d;
END_VAR
// check if to hold the command joint position unchanged
m_holdLastCmds := checkToHoldLastCmds(i_slaveArm);

//init
SUPER^.Init(i_slaveArm,r_slaveArmCtrlCmd);
END_METHOD

END_FUNCTION_BLOCK

// ---- FBs_SlaveControllers/FB_SlaveCtrlGraCali.TcPOU
// Brief: Slave Arm Gravity Calibration
FUNCTION_BLOCK PUBLIC FB_SlaveCtrlGraCali EXTENDS FB_SlaveArmCtrlBase
VAR_INPUT
END_VAR
VAR_OUTPUT
END_VAR
VAR
// cali trajectory
	m_caliMotionSegs :INT :=3;
	m_graCaliTraj:ARRAY [1..3, 1..g_sJntNum] OF LREAL:=
		[-pi/6, -PI/2+pi/6, 0.5, 	5(-pi/3),
		 pi/6, 	-PI/2-pi/4, 0.3, 	5(0),
		 -pi/6, -PI/2+pi/6, 0.5, 	5(-pi/3)];
		 
	m_caliMaxjntVel:Vec8d:=[2(2.5*g_deg2Rad), 0.01, 5(2.5*g_deg2Rad)];
	m_caliMaxjntAcc:Vec8d:=[8(0.5)];
	m_caliMaxjntJerk:Vec8d:=[8(2.0)];
	
	m_caliTrajIdx: INT := 1;
	m_caliPlanner: ARRAY[1..3] OF FB_TrajMoveJ;
	
END_VAR

// override this function in each exact controller
METHOD PROTECTED calcCmdJntPos : BOOL
VAR_IN_OUT CONSTANT
	i_endoscopePose : ST_Frame;
	i_masterStatus :ST_MasterStatus;
	i_setupStatus: ST_SetupStatus;
	i_slaveArm :FB_SlaveArm;
END_VAR


VAR 
	i :INT;
	curJntVel :Vec8d;
END_VAR
// check if planner is ready
IF m_caliPlanner[m_caliTrajIdx].isGene = FALSE THEN
	calcCmdJntPos:=FALSE;
	RETURN;
END_IF

// traj plan
calcCmdJntPos :=m_caliPlanner[m_caliTrajIdx].evaluate(m_timePeriod, jntPos=> m_cmdJntPos, jntVel=>m_cmdJntVel, jntAcc=> m_cmdJntAcc);

// check if to transit to next segment
curJntVel :=i_slaveArm.curJntVel;
IF(m_timePeriod > m_caliPlanner[m_caliTrajIdx].duration  AND norm(curJntVel)<7*GVL_SlaveControlParameters.g_jntStaticVelThres) THEN
	m_caliTrajIdx:=m_caliTrajIdx+1;
	m_timePeriod:=0;
END_IF

// check if to terminated
IF(m_caliTrajIdx > m_caliMotionSegs) THEN
	m_isFinished:=TRUE;
END_IF
END_METHOD

METHOD PUBLIC init : BOOL
VAR_IN_OUT CONSTANT
	i_slaveArm	:FB_SlaveArm;
END_VAR
VAR_IN_OUT 
	r_slaveArmCtrlCmd :ST_SlaveArmCtrlCmds;
END_VAR

VAR
	i,j :INT;
	initJntPos,startJntPos,endJntPos :Vec8d;

END_VAR
SUPER^.Init(i_slaveArm,r_slaveArmCtrlCmd);
m_caliTrajIdx :=1;
m_jntOPMode := g_slaveAllPosTrqMode;

// traj plan
// fisrt segment
initJntPos:=i_slaveArm.curJntPos;
startJntPos:=initJntPos;
endJntPos:=startJntPos;
FOR j:=1 TO g_sJntNum DO 
	IF j>3 THEN
		endJntPos[j]:=initJntPos[j]+ m_graCaliTraj[1,j];
	ELSE
		endJntPos[j]:=m_graCaliTraj[1,j];
	END_IF
END_FOR
m_caliPlanner[1].init(startJntPos,endJntPos,m_caliMaxjntVel, m_caliMaxJntAcc, m_caliMaxJntJerk);

// other segments
FOR i:=2 TO m_caliMotionSegs DO 
	startJntPos := endJntPos;
	FOR j:=1 TO g_sJntNum DO 
		IF j>3 THEN
			endJntPos[j]:=initJntPos[j]+ m_graCaliTraj[i,j];
		ELSE
			endJntPos[j]:=m_graCaliTraj[i,j];
		END_IF
	END_FOR
	m_caliPlanner[i].init(startJntPos,endJntPos,m_caliMaxjntVel, m_caliMaxJntAcc, m_caliMaxJntJerk);
END_FOR

// update commands to arm
copyCmds(r_slaveArmCtrlCmd);
END_METHOD

END_FUNCTION_BLOCK

// ---- FBs_SlaveControllers/FB_SlaveCtrlTest.TcPOU
// Brief: Slave Arm test
FUNCTION_BLOCK PUBLIC FB_SlaveCtrlTest EXTENDS FB_SlaveArmCtrlBase
VAR_INPUT
END_VAR
VAR_OUTPUT
END_VAR
VAR
// ################ variables for single DH  joint test ##################
	m_enableFrictionComp :BOOL :=false;
	m_freqTestFlag :BOOL:=FALSE;
	m_initJntPos :Vec8d;
	m_initDHJntPos :Vec6d;
	m_cmdDHJntPos :Vec6d;
	m_cmdDHJntVel :Vec6d;
	m_jntMotionFreq :Vec6d :=[0.2, 0.2, 0.1, 3(0.1)];
	m_jntMotionRange :Vec6d :=[pi/6, pi/6, 0.1, 3(pi/6)];
	m_testJntIdx :INT :=1;
	m_gripperAngle : LREAL :=0;
	m_gripForceLevel :LREAL :=0;
	m_lastCmdJntPos :Vec8d ;
	
	m_stepTestFlag :BOOL :=FALSE;
	m_jntStep : LREAL := 5*g_deg2Rad;
	
	// instrument controller
	m_instruController : FB_BasicInstruControl;
	m_instruCmdJntPos,m_instruCmdJntVel : Vec5d;
	m_instruCmdJntTrq :Vec5d;
	
	
	m_errCmdPos, m_errCurPos :LREAL;
	m_errPosIdx : INT;
	
	// instrument rotation test
	m_instruRotTest :BOOL :=FALSE;
	m_instruRotOTG : FB_secOrdTrajFilter;
	m_slaveOriginPose : ST_Frame;
	m_slaveCmdPose : ST_Frame;
	m_instruRotAxis :Vec3d := [0, 0, 1];
	
	// friciton test
	m_staticFrictionTest : BOOL := FALSE;
	m_colFrictionTest :BOOL :=FALSE;
	
	
//####################################################################

END_VAR

METHOD PROTECTED calcCmdJntPos : BOOL
VAR_IN_OUT CONSTANT
	i_endoscopePose : ST_Frame;
	i_masterStatus :ST_MasterStatus;
	i_setupStatus: ST_SetupStatus;
	i_slaveArm :FB_SlaveArm;
END_VAR

VAR 
	i:INT :=0;
	errThres :LREAL;
	m_masterGripAngle: INT;
	instruRotAng:REAL;
	instruRotMat:Mat3d;
	slavePosErr:Vec3d;
	tmpMat3d:Mat3d;
	slaveRotErr :Mat3d;
	errAngle:LREAL;
	errAxisLocal,errAxis:Vec3d;
	slaveCmdVel, slaveCmdWVel:Vec3d;
	slaveTrackTwist:Vec6d;
	cmdVelScale :REAL:=1;
	invJaco :Mat6d;
	simDHJointVel:Vec6d;
	DHJntCmdDeltaPos:Vec6d;
END_VAR
IF i_slaveArm.instruOn THEN
	calcCmdJntPos_withInstru(i_endoscopePose,i_masterStatus,i_setupStatus,i_slaveArm);
ELSE
	calcCmdJntPos_noInstru(i_endoscopePose,i_masterStatus,i_setupStatus,i_slaveArm);
END_IF
END_METHOD

METHOD PROTECTED calcCmdJntPos_noInstru : BOOL
VAR_IN_OUT CONSTANT
	i_endoscopePose : ST_Frame;
	i_masterStatus :ST_MasterStatus;
	i_setupStatus: ST_SetupStatus;
	i_slaveArm :FB_SlaveArm;
END_VAR

VAR 
	i:INT :=0;
	errThres :LREAL;
	m_masterGripAngle: INT;
	instruRotAng:REAL;
	instruRotMat:Mat3d;
	slavePosErr:Vec3d;
	tmpMat3d:Mat3d;
	slaveRotErr :Mat3d;
	errAngle:LREAL;
	errAxisLocal,errAxis:Vec3d;
	slaveCmdVel, slaveCmdWVel:Vec3d;
	slaveTrackTwist:Vec6d;
	cmdVelScale :REAL:=1;
	invJaco :Mat6d;
	simDHJointVel:Vec6d;
	DHJntCmdDeltaPos:Vec6d;
END_VAR
// Just for joint controller test
IF m_testJntIdx >=1 AND m_testJntIdx <=8 THEN
	IF m_freqTestFlag THEN 
		m_cmdJntPos[m_testJntIdx]:=m_initJntPos[m_testJntIdx]+m_jntMotionRange[m_testJntIdx]/2
										+0.5*m_jntMotionRange[m_testJntIdx]*SIN(2*pi*m_jntMotionFreq[m_testJntIdx]*m_timePeriod-pi/2);
		m_cmdJntVel[m_testJntIdx]:=0.5*m_jntMotionRange[m_testJntIdx]*2*pi*m_jntMotionFreq[m_testJntIdx]*COS(2*pi*m_jntMotionFreq[m_testJntIdx]*m_timePeriod-pi/2);
	ELSIF m_stepTestFlag THEN
		m_cmdJntPos[m_testJntIdx]:=m_initJntPos[m_testJntIdx]+m_jntStep;
	ELSIF m_colFrictionTest THEN
		m_cmdJntPos[m_testJntIdx]:=m_cmdJntPos[m_testJntIdx]+ g_slaveArmCtrlCycleTime * 45*g_deg2rad;
	ELSIF m_staticFrictionTest THEN
		m_jntOPMode[m_testJntIdx] := DriverOPMode_Trq;
		m_cmdJntTrq[m_testJntIdx]:=m_cmdJntTrq[m_testJntIdx] + g_slaveArmCtrlCycleTime*2/1000.0*GVL_SlaveMotorParameters.g_motorTrqConst[m_testJntIdx]*GVL_SlaveMotorParameters.g_motorReduction[m_testJntIdx];
		m_cmdJntPos[m_testJntIdx]:=i_slaveArm.curJntPos[m_testJntIdx];
		IF ABS(i_slaveArm.curJntVel[m_testJntIdx])>5*g_deg2rad THEN
			m_jntOPMode[m_testJntIdx] := DriverOPMode_PosTrq;
			m_staticFrictionTest:=FALSE;
		END_IF
	ELSE
		m_timePeriod:=0;
		m_cmdJntTrq[m_testJntIdx]:=0;
	END_IF
	
END_IF


m_lastCmdJntPos:=m_cmdJntPos;

FOR i:=1 TO 3 DO 
	IF i=3 THEN
		errThres := 0.01;
	ELSE
		errThres :=5*g_deg2rad;
	END_IF
	
	IF ABS(m_cmdJntPos[i]-i_slaveArm.curJntPos[i])>errThres THEN
		m_isFinished:=TRUE;
		m_errPosIdx:=i;
		m_errCmdPos:=m_cmdJntPos[i];
		m_errCurPos :=i_slaveArm.curJntPos[i];
	END_IF
	
END_FOR
END_METHOD

METHOD PROTECTED calcCmdJntPos_withInstru : BOOL
VAR_IN_OUT CONSTANT
	i_endoscopePose : ST_Frame;
	i_masterStatus :ST_MasterStatus;
	i_setupStatus: ST_SetupStatus;
	i_slaveArm :FB_SlaveArm;
END_VAR

VAR 
	i:INT :=0;
	errThres :LREAL;
	m_masterGripAngle: INT;
	instruRotAng:REAL;
	instruRotMat:Mat3d;
	slavePosErr:Vec3d;
	tmpMat3d:Mat3d;
	slaveRotErr :Mat3d;
	errAngle:LREAL;
	errAxisLocal,errAxis:Vec3d;
	slaveCmdVel, slaveCmdWVel:Vec3d;
	slaveTrackTwist:Vec6d;
	cmdVelScale :REAL:=1;
	invJaco :Mat6d;
	simDHJointVel:Vec6d;
	DHJntCmdDeltaPos:Vec6d;
END_VAR
// Just for joint controller test
IF m_testJntIdx >=1 AND m_testJntIdx <=6 THEN
	IF m_freqTestFlag THEN 
		m_cmdDHJntPos[m_testJntIdx]:=m_initDHJntPos[m_testJntIdx]+m_jntMotionRange[m_testJntIdx]/2
										+0.5*m_jntMotionRange[m_testJntIdx]*SIN(2*pi*m_jntMotionFreq[m_testJntIdx]*m_timePeriod-pi/2);
		m_cmdDHJntVel[m_testJntIdx]:=0.5*m_jntMotionRange[m_testJntIdx]*2*pi*m_jntMotionFreq[m_testJntIdx]*COS(2*pi*m_jntMotionFreq[m_testJntIdx]*m_timePeriod-pi/2);
	ELSIF m_stepTestFlag THEN
		m_cmdDHJntPos[m_testJntIdx]:=m_initDHJntPos[m_testJntIdx]+m_jntStep;
	ELSE
		m_timePeriod:=0;
	END_IF
	
END_IF

// instrument rotation test
IF m_instruRotTest AND NOT(m_freqTestFlag) AND NOT(m_stepTestFlag) THEN
	m_instruRotOTG.run(m_jntStep,0.0, o_cmdAcc=>,o_cmdVel=>,o_cmdPos=> instruRotAng);
	instruRotMat :=  angAxis2Rot(instruRotAng,m_instruRotAxis);
	matMultiply(m_slaveOriginPose.m_rot, instruRotMat,m_slaveCmdPose.m_rot );
	
		
	// compute pose error
	vecSub(m_slaveCmdPose.m_pos, i_slaveArm.simCartPose.m_pos, slavePosErr);
	matTranspose(i_slaveArm.simCartPose.m_rot, tmpMat3d);
	matMultiply(tmpMat3d, m_slaveCmdPose.m_rot, slaveRotErr);
	rot2AngAxis(slaveRotErr, angle=>errAngle, axis=>errAxisLocal);
	matMultiVec(i_slaveArm.simCartPose.m_rot, errAxisLocal, errAxis);
	
	// pose track control
	vecMultiNum(slavePosErr, g_slaveArmCtrlFreq, slaveCmdVel);
	vecMultiNum(errAxis, errAngle*g_slaveArmCtrlFreq, slaveCmdWVel);
	FOR i:=1 TO 3 DO 
		slaveTrackTwist[i] := slaveCmdVel[i];
		slaveTrackTwist[i+3] := slaveCmdWVel[i];
	END_FOR
	
	// compute command velocity for DH joints
	invJaco := i_slaveArm.simJacoInv;
	matMultiVec(invJaco, slaveTrackTwist, simDHJointVel);
	
	// limit DH joints velocity 
	cmdVelScale := 1;
	FOR i:=1 TO g_cartDofs DO 
		cmdVelScale:=MAX(cmdVelScale, ABS(simDHJointVel[i]/GVL_SlaveMotorParameters.g_maxJntVel[i]));
	END_FOR
	vecSelfMultiNum(simDHJointVel, 1.0/cmdVelScale);
	
	// integrate command DH joint position
	vecMultiNum(simDHJointVel, g_slaveArmCtrlCycleTime, DHJntCmdDeltaPos);
	vecSelfAdd(m_cmdDHJntPos, DHJntCmdDeltaPos);
	
ELSE
	m_slaveOriginPose := i_slaveArm.simCartPose;
	m_slaveCmdPose := m_slaveOriginPose;
END_IF

// calculate target motor joint position from DH joint position
i_slaveArm.instrument.instruIK(m_cmdDHJntPos,m_gripperAngle, o_jntPos=>m_cmdJntPos);
//m_cmdJntPos[4]:=m_originalJntPos[4];
//m_cmdJntPos[5]:=m_originalJntPos[5];
//m_cmdJntPos[6]:=m_originalJntPos[6];
//m_cmdJntPos[7]:=m_originalJntPos[7];
//m_cmdJntPos[8]:=m_originalJntPos[8];

IF m_freqTestFlag THEN 
	vecSub(m_cmdJntPos, m_lastCmdJntPos, m_cmdJntVel);
	vecSelfMultiNum(m_cmdJntVel, g_slaveArmCtrlFreq);
ELSE
	m_cmdJntVel:=g_zeroVec8d;
END_IF
m_lastCmdJntPos:=m_cmdJntPos;

FOR i:=1 TO 3 DO 
	IF i=3 THEN
		errThres := 0.01;
	ELSE
		errThres :=5*g_deg2rad;
	END_IF
	
	IF ABS(m_cmdDHJntPos[i]-i_slaveArm.curDHJntPos[i])>errThres THEN
		m_isFinished:=TRUE;
		m_errPosIdx:=i;
		m_errCmdPos:=m_cmdJntPos[i];
		m_errCurPos :=i_slaveArm.curJntPos[i];
	END_IF
	
END_FOR
END_METHOD

// override this function in each exact controller
METHOD PROTECTED calcCmdJntTrq : BOOL
VAR_IN_OUT CONSTANT
	i_endoscopePose : ST_Frame;
	i_masterStatus :ST_MasterStatus;
	i_setupStatus: ST_SetupStatus;
	i_slaveArm :FB_SlaveArm;
END_VAR

VAR 
	nullspaceMat :Mat7d;
	ctrlTrq : Vec7d;
	i : int ;
END_VAR
IF not(i_slaveArm.instruOn) THEN
	RETURN;
END_IF

// set joint torque to zero in default
m_cmdJntTrq := g_zeroVec8d;

// instrument joint control

FOR i:=1 TO 5 DO 
	m_instruCmdJntPos[i]:=m_cmdJntPos[i+3];
	m_instruCmdJntVel[i]:=m_cmdJntVel[i+3];
END_FOR
m_instruController.run(m_instruCmdJntPos,m_instruCmdJntVel, m_cmdDHJntPos[6], m_cmdDHJntVel[6], m_gripForceLevel, i_slaveArm, o_cmdJntTrq=>m_instruCmdJntTrq);

FOR i:=1 TO 5 DO
	m_cmdJntTrq[i+3]:=m_instruCmdJntTrq[i];
END_FOR

// add friction
IF m_enableFrictionComp THEN
	enableFrictionCompensation(i_slaveArm);
END_IF
END_METHOD

METHOD PUBLIC init : BOOL
VAR_IN_OUT CONSTANT
	i_slaveArm	:FB_SlaveArm;
END_VAR
VAR_IN_OUT 
	r_slaveArmCtrlCmd :ST_SlaveArmCtrlCmds;
END_VAR
SUPER^.Init(i_slaveArm,r_slaveArmCtrlCmd);
m_lastCmdJntPos:=m_cmdJntPos;
m_jntOPMode[1] := DriverOPMode_PosTrq;
m_jntOPMode[2] := DriverOPMode_PosTrq;
m_jntOPMode[3] := DriverOPMode_PosTrq;
IF i_slaveArm.instruOn THEN
	m_jntOPMode[4] := DriverOPMode_Trq;
	m_jntOPMode[5] := DriverOPMode_Trq;
	m_jntOPMode[6] := DriverOPMode_Trq;
	m_jntOPMode[7] := DriverOPMode_Trq;
	m_jntOPMode[8] := DriverOPMode_Trq;

ELSE
	m_jntOPMode[4] := DriverOPMode_PosTrq;
	m_jntOPMode[5] := DriverOPMode_PosTrq;
	m_jntOPMode[6] := DriverOPMode_PosTrq;
	m_jntOPMode[7] := DriverOPMode_PosTrq;
	m_jntOPMode[8] := DriverOPMode_PosTrq;
END_IF


m_initDHJntPos :=i_slaveArm.curDHJntPos;
m_initJntPos := i_slaveArm.curJntPos;
m_cmdDHJntPos :=m_initDHJntPos;
m_cmdDHJntVel :=g_zeroVec6d;
m_gripperAngle := i_slaveArm.curGripAngle;

// init instrument controller
m_instruController.init(i_slaveArm);

m_instruRotOTG.init(0, 0,1, 2, g_slaveArmCtrlCycleTime);


// update commands to arm
copyCmds(r_slaveArmCtrlCmd);
END_METHOD

END_FUNCTION_BLOCK

// ---- FBs_SlaveControllers/FB_SlaveCtrlInstruRetract.TcPOU
// Brief: Slave Arm joint3 retract to up limit
FUNCTION_BLOCK PUBLIC FB_SlaveCtrlInstruRetract EXTENDS FB_SlaveArmCtrlBase
VAR_INPUT
END_VAR
VAR_OUTPUT
END_VAR
VAR
	// wait time before retract, ensure instruments is removed 
	m_waitTime :LREAL :=2.0;
		
	// motion planning
	m_jnt3OTG : FB_secOrdTrajFilter;
	m_jnt3TargetPos :LREAL;
	m_retractVel: LREAL:= 0.1;
	m_retractAcc: LREAL:= 0.2;
	
	// instrument joint motion planning
	m_instruJntOTG :ARRAY[1..5] OF FB_secOrdTrajFilter;
	m_instruJntTargetPos :Vec5d;
	m_instruJntVel :LREAL := 2*PI;
	m_instruJntAcc : LREAL := 4*PI;
	
	
END_VAR

// override this function in each exact controller
METHOD PROTECTED calcCmdJntPos : BOOL
VAR_IN_OUT CONSTANT
	i_endoscopePose : ST_Frame;
	i_masterStatus :ST_MasterStatus;
	i_setupStatus: ST_SetupStatus;
	i_slaveArm :FB_SlaveArm;
END_VAR

VAR 
	i :INT;
	trackErr:LREAL;
	curJntVel:Vec8d;
END_VAR
// if instrument is on again, wait and re-plan the traj
IF i_slaveArm.instruNear THEN
	m_cmdJntVel:=g_zeroVec8d;
	m_cmdJntAcc := g_zeroVec8d;
	
	// init traj filter
	m_jnt3OTG.init(m_cmdJntPos[3], 0, m_retractVel, m_retractAcc, g_slaveArmCtrlCycleTime);
	FOR i:=1 TO 5 DO
		m_instruJntOTG[i].init(m_cmdJntPos[i+3], 0,m_instruJntVel, m_instruJntAcc, g_slaveArmCtrlCycleTime);
	END_FOR

	m_timePeriod := 0;
	RETURN;
END_IF

// wait
IF m_timePeriod< m_waitTime THEN
	RETURN;
END_IF

// traj plan
m_jnt3OTG.run(m_jnt3TargetPos, 0.0, o_cmdAcc=>m_cmdJntAcc[3],o_cmdVel=>m_cmdJntVel[3],o_cmdPos=>m_cmdJntPos[3]);
FOR i:=1 TO 5 DO
	m_instruJntOTG[i].run(m_instruJntTargetPos[i], 0.0, o_cmdAcc=>m_cmdJntAcc[i+3],o_cmdVel=>m_cmdJntVel[i+3],o_cmdPos=>m_cmdJntPos[i+3]);
END_FOR

// reach target check
trackErr :=0;
FOR i:=1 TO 5 DO 
	trackErr := MAX(trackErr, ABS(m_cmdJntPos[i+3]-m_instruJntTargetPos[i]));
END_FOR
curJntVel := i_slaveArm.curJntVel;
m_isFinished := (ABS(m_cmdJntPos[3] - m_jnt3TargetPos) <g_cartCtrlPosTolLow AND trackErr < g_jntCtrlAngTolLoW 
			AND norm(curJntVel) <g_jntStaticVelThres);
END_METHOD

METHOD PUBLIC init : BOOL
VAR_IN_OUT CONSTANT
	i_slaveArm	:FB_SlaveArm;
END_VAR
VAR_IN_OUT 
	r_slaveArmCtrlCmd :ST_SlaveArmCtrlCmds;
END_VAR

VAR
	i:INT;
	cycleNum:LREAL;
END_VAR
// check if to hold the command joint position unchanged
m_holdLastCmds := checkToHoldLastCmds(i_slaveArm);

SUPER^.Init(i_slaveArm,r_slaveArmCtrlCmd);

// decide target position
m_jnt3TargetPos := GVL_SlaveMotorParameters.g_maxDHJntPos[3];

